LIN {X 0,Y 178.864,Z 372.474,A -85,B 0,C 180,E1 -23549.283,E2 -23549.283} C_VEL
LIN {X 0,Y 171.89,Z 372.083,A -85,B 0,C 180,E1 -23553.272,E2 -23553.272} C_VEL
LIN {X 0,Y 166.102,Z 370.53,A -85,B 0,C 180,E1 -23557.617,E2 -23557.617} C_VEL
LIN {X 0,Y 161.684,Z 367.817,A -85,B 0,C 180,E1 -23562.286,E2 -23562.286} C_VEL
LIN {X 0,Y 158.988,Z 364.935,A -85,B 0,C 180,E1 -23565.929,E2 -23565.929} C_VEL
LIN {X 0,Y 156.894,Z 359.998,A -85,B 0,C 180,E1 -23570.999,E2 -23570.999} C_VEL
LIN {X 0,Y 156.126,Z 355.356,A -85,B 0,C 180,E1 -23574.835,E2 -23574.835} C_VEL
LIN {X 0,Y 155.711,Z 348.695,A -85,B 0,C 180,E1 -23579.354,E2 -23579.354} C_VEL
LIN {X 0,Y 155.836,Z 341.725,A -85,B 0,C 180,E1 -23583.232,E2 -23583.232} C_VEL
LIN {X 0,Y 156.247,Z 333.011,A -85,B 0,C 180,E1 -23587.197,E2 -23587.197} C_VEL
LIN {X 0,Y 157.032,Z 322.982,A -85,B 0,C 180,E1 -23590.965,E2 -23590.965} C_VEL
LIN {X 0,Y 158.084,Z 311.456,A -85,B 0,C 180,E1 -23594.482,E2 -23594.482} C_VEL
LIN {X 0,Y 159.277,Z 300.027,A -85,B 0,C 180,E1 -23597.328,E2 -23597.328} C_VEL
LIN {X 0,Y 160.585,Z 287.52,A -85,B 0,C 180,E1 -23599.827,E2 -23599.827} C_VEL
LIN {X 0,Y 159.751,Z 280.238,A -85,B 0,C 180,E1 -23601.02,E2 -23601.02} C_VEL
LIN {X 0,Y 158.066,Z 266.61,A -85,B 0,C 180,E1 -23602.867,E2 -23602.867} C_VEL
LIN {X 0,Y 157.49,Z 258.741,A -85,B 0,C 180,E1 -23603.767,E2 -23603.767} C_VEL
LIN {X 0,Y 158.382,Z 249.573,A -85,B 0,C 180,E1 -23609.948,E2 -23609.948} C_VEL
LIN {X 0,Y 159.359,Z 242.124,A -85,B 0,C 180,E1 -23614.982,E2 -23614.982} C_VEL
LIN {X 0,Y 159.793,Z 237.68,A -85,B 0,C 180,E1 -23618.007,E2 -23618.007} C_VEL
LIN {X 0,Y 159.018,Z 232.396,A -85,B 0,C 180,E1 -23621.843,E2 -23621.843} C_VEL
LIN {X 0,Y 159.402,Z 233.851,A -85,B 0,C 180,E1 -23625.131,E2 -23625.131} C_VEL
LIN {X 0,Y 159.637,Z 235.642,A -85,B 0,C 180,E1 -23628.668,E2 -23628.668} C_VEL
LIN {X 0,Y 160.053,Z 238.877,A -85,B 0,C 180,E1 -23634.376,E2 -23634.376} C_VEL
LIN {X 0,Y 161.694,Z 242.388,A -85,B 0,C 180,E1 -23635.252,E2 -23635.252} C_VEL
LIN {X 0,Y 165.253,Z 249.918,A -85,B 0,C 180,E1 -23637.133,E2 -23637.133} C_VEL
LIN {X 0,Y 167.935,Z 257.855,A -85,B 0,C 180,E1 -23639.086,E2 -23639.086} C_VEL
LIN {X 0,Y 169.717,Z 265.352,A -85,B 0,C 180,E1 -23641.054,E2 -23641.054} C_VEL
LIN {X 0,Y 170.772,Z 272.517,A -85,B 0,C 180,E1 -23643.08,E2 -23643.08} C_VEL
LIN {X 0,Y 171.198,Z 278.169,A -85,B 0,C 180,E1 -23644.84,E2 -23644.84} C_VEL
LIN {X 0,Y 170.665,Z 280.993,A -85,B 0,C 180,E1 -23645.679,E2 -23645.679} C_VEL
LIN {X 0,Y 167.855,Z 289.578,A -85,B 0,C 180,E1 -23648.506,E2 -23648.506} C_VEL
LIN {X 0,Y 165.094,Z 296.179,A -85,B 0,C 180,E1 -23651.378,E2 -23651.378} C_VEL
LIN {X 0,Y 163.429,Z 300.329,A -85,B 0,C 180,E1 -23653.765,E2 -23653.765} C_VEL
LIN {X 0,Y 161.928,Z 303.706,A -85,B 0,C 180,E1 -23656.186,E2 -23656.186} C_VEL
LIN {X 0,Y 160.418,Z 307.486,A -85,B 0,C 180,E1 -23659.904,E2 -23659.904} C_VEL
LIN {X 0,Y 159.37,Z 309.319,A -85,B 0,C 180,E1 -23662.394,E2 -23662.394} C_VEL
LIN {X 0,Y 158.847,Z 310.546,A -85,B 0,C 180,E1 -23664.92,E2 -23664.92} C_VEL
LIN {X 0,Y 158.433,Z 311.303,A -85,B 0,C 180,E1 -23667.454,E2 -23667.454} C_VEL
LIN {X 0,Y 158.279,Z 311.577,A -85,B 0,C 180,E1 -23669.997,E2 -23669.997} C_VEL
LIN {X 0,Y 158.432,Z 311.335,A -85,B 0,C 180,E1 -23672.539,E2 -23672.539} C_VEL
LIN {X 0,Y 158.845,Z 310.622,A -85,B 0,C 180,E1 -23675.073,E2 -23675.073} C_VEL
LIN {X 0,Y 159.367,Z 309.426,A -85,B 0,C 180,E1 -23677.599,E2 -23677.599} C_VEL
LIN {X 0,Y 160.955,Z 306.53,A -85,B 0,C 180,E1 -23681.328,E2 -23681.328} C_VEL
LIN {X 0,Y 162.457,Z 302.377,A -85,B 0,C 180,E1 -23685.041,E2 -23685.041} C_VEL
LIN {X 0,Y 163.482,Z 300.591,A -85,B 0,C 180,E1 -23686.223,E2 -23686.223} C_VEL
LIN {X 0,Y 165.079,Z 296.507,A -85,B 0,C 180,E1 -23688.617,E2 -23688.617} C_VEL
LIN {X 0,Y 167.817,Z 289.962,A -85,B 0,C 180,E1 -23691.493,E2 -23691.493} C_VEL
LIN {X 0,Y 170.602,Z 281.568,A -85,B 0,C 180,E1 -23694.324,E2 -23694.324} C_VEL
LIN {X 0,Y 171.271,Z 277.73,A -85,B 0,C 180,E1 -23695.476,E2 -23695.476} C_VEL
LIN {X 0,Y 170.427,Z 269.133,A -85,B 0,C 180,E1 -23698.096,E2 -23698.096} C_VEL
LIN {X 0,Y 168.581,Z 260.042,A -85,B 0,C 180,E1 -23700.542,E2 -23700.542} C_VEL
LIN {X 0,Y 165.775,Z 251.147,A -85,B 0,C 180,E1 -23702.753,E2 -23702.753} C_VEL
LIN {X 0,Y 161.837,Z 242.466,A -85,B 0,C 180,E1 -23704.901,E2 -23704.901} C_VEL
LIN {X 0,Y 160.31,Z 239.516,A -85,B 0,C 180,E1 -23705.627,E2 -23705.627} C_VEL
LIN {X 0,Y 160.14,Z 238.936,A -85,B 0,C 180,E1 -23705.743,E2 -23705.743} C_VEL
LIN {X 0,Y 159.65,Z 235.706,A -85,B 0,C 180,E1 -23711.551,E2 -23711.551} C_VEL
LIN {X 0,Y 159.33,Z 233.908,A -85,B 0,C 180,E1 -23715.109,E2 -23715.109} C_VEL
LIN {X 0,Y 159.092,Z 232.317,A -85,B 0,C 180,E1 -23718.67,E2 -23718.67} C_VEL
LIN {X 0,Y 158.736,Z 230.624,A -85,B 0,C 180,E1 -23722.833,E2 -23722.833} C_VEL
LIN {X 0,Y 158.461,Z 228.914,A -85,B 0,C 180,E1 -23727.844,E2 -23727.844} C_VEL
LIN {X 0,Y 158.156,Z 227.327,A -85,B 0,C 180,E1 -23733.617,E2 -23733.617} C_VEL
LIN {X 0,Y 157.925,Z 226.263,A -85,B 0,C 180,E1 -23739.144,E2 -23739.144} C_VEL
LIN {X 0,Y 157.872,Z 225.638,A -85,B 0,C 180,E1 -23744.508,E2 -23744.508} C_VEL
LIN {X 0,Y 158.084,Z 225.448,A -85,B 0,C 180,E1 -23749.756,E2 -23749.756} C_VEL
LIN {X 0,Y 158.195,Z 225.509,A -85,B 0,C 180,E1 -23752.341,E2 -23752.341} C_VEL
LIN {X 0,Y 158.794,Z 226.144,A -85,B 0,C 180,E1 -23760,E2 -23760} C_VEL
LIN {X 0,Y 158.687,Z 227.58,A -85,B 0,C 180,E1 -23765.082,E2 -23765.082} C_VEL
LIN {X 0,Y 159.105,Z 229.328,A -85,B 0,C 180,E1 -23770.177,E2 -23770.177} C_VEL
LIN {X 0,Y 159.387,Z 231.672,A -85,B 0,C 180,E1 -23775.341,E2 -23775.341} C_VEL
LIN {X 0,Y 159.941,Z 234.494,A -85,B 0,C 180,E1 -23780.581,E2 -23780.581} C_VEL
LIN {X 0,Y 160.713,Z 237.968,A -85,B 0,C 180,E1 -23785.932,E2 -23785.932} C_VEL
LIN {X 0,Y 161.422,Z 240.536,A -85,B 0,C 180,E1 -23789.46,E2 -23789.46} C_VEL
LIN {X 0,Y 162.358,Z 244.484,A -85,B 0,C 180,E1 -23794.245,E2 -23794.245} C_VEL
LIN {X 0,Y 163.242,Z 249.108,A -85,B 0,C 180,E1 -23799.206,E2 -23799.206} C_VEL
LIN {X 0,Y 164.036,Z 253.296,A -85,B 0,C 180,E1 -23803.276,E2 -23803.276} C_VEL
LIN {X 0,Y 165.228,Z 258.701,A -85,B 0,C 180,E1 -23808.211,E2 -23808.211} C_VEL
LIN {X 0,Y 165.717,Z 261.5,A -85,B 0,C 180,E1 -23810.491,E2 -23810.491} C_VEL
LIN {X 0,Y 167.275,Z 265.557,A -85,B 0,C 180,E1 -23811.212,E2 -23811.212} C_VEL
LIN {X 0,Y 167.835,Z 268.967,A -85,B 0,C 180,E1 -23811.673,E2 -23811.673} C_VEL
LIN {X 0,Y 168.302,Z 280.321,A -85,B 0,C 180,E1 -23813.191,E2 -23813.191} C_VEL
LIN {X 0,Y 167.94,Z 290.791,A -85,B 0,C 180,E1 -23814.876,E2 -23814.876} C_VEL
LIN {X 0,Y 166.952,Z 302.091,A -85,B 0,C 180,E1 -23817.146,E2 -23817.146} C_VEL
LIN {X 0,Y 165.032,Z 313.463,A -85,B 0,C 180,E1 -23819.979,E2 -23819.979} C_VEL
LIN {X 0,Y 163.62,Z 321.527,A -85,B 0,C 180,E1 -23822.504,E2 -23822.504} C_VEL
LIN {X 0,Y 162.576,Z 326.775,A -85,B 0,C 180,E1 -23824.391,E2 -23824.391} C_VEL
LIN {X 0,Y 159.816,Z 335.261,A -85,B 0,C 180,E1 -23828.075,E2 -23828.075} C_VEL
LIN {X 0,Y 157.929,Z 341.848,A -85,B 0,C 180,E1 -23831.854,E2 -23831.854} C_VEL
LIN {X 0,Y 156.88,Z 347.042,A -85,B 0,C 180,E1 -23835.739,E2 -23835.739} C_VEL
LIN {X 0,Y 156.611,Z 350.924,A -85,B 0,C 180,E1 -23839.663,E2 -23839.663} C_VEL
LIN {X 0,Y 156.875,Z 352.842,A -85,B 0,C 180,E1 -23842.28,E2 -23842.28} C_VEL
LIN {X 0,Y 157.572,Z 354.473,A -85,B 0,C 180,E1 -23845.046,E2 -23845.046} C_VEL
LIN {X 0,Y 157.668,Z 360.13,A -85,B 0,C 180,E1 -23848.088,E2 -23848.088} C_VEL
LIN {X 0,Y 157.721,Z 364.985,A -85,B 0,C 180,E1 -23851.28,E2 -23851.28} C_VEL
LIN {X 0,Y 157.19,Z 368.04,A -85,B 0,C 180,E1 -23853.849,E2 -23853.849} C_VEL
LIN {X 0,Y 156.604,Z 372.902,A -85,B 0,C 180,E1 -23859.139,E2 -23859.139} C_VEL
LIN {X 0,Y 157.016,Z 375.5,A -85,B 0,C 180,E1 -23862.936,E2 -23862.936} C_VEL
LIN {X 0,Y 158.818,Z 378.029,A -85,B 0,C 180,E1 -23868.048,E2 -23868.048} C_VEL
LIN {X 0,Y 162.378,Z 379.502,A -85,B 0,C 180,E1 -23872.929,E2 -23872.929} C_VEL
LIN {X 0,Y 167.343,Z 379.897,A -85,B 0,C 180,E1 -23877.518,E2 -23877.518} C_VEL
LIN {X 0,Y 173.897,Z 379.136,A -85,B 0,C 180,E1 -23882.062,E2 -23882.062} C_VEL
LIN {X 0,Y 176.385,Z 378.542,A -85,B 0,C 180,E1 -23883.806,E2 -23883.806} C_VEL
LIN {X 0,Y 182.265,Z 376.171,A -85,B 0,C 180,E1 -23889.128,E2 -23889.128} C_VEL
LIN {X 0,Y 185.289,Z 375.099,A -85,B 0,C 180,E1 -23890.661,E2 -23890.661} C_VEL
LIN {X 0,Y 186.544,Z 374.692,A -85,B 0,C 180,E1 -23891.107,E2 -23891.107} C_VEL
LIN {X 0,Y 196.969,Z 371.002,A -85,B 0,C 180,E1 -23894.092,E2 -23894.092} C_VEL
LIN {X 0,Y 206.383,Z 366.992,A -85,B 0,C 180,E1 -23896.276,E2 -23896.276} C_VEL
LIN {X 0,Y 206.868,Z 366.673,A -85,B 0,C 180,E1 -23896.802,E2 -23896.802} C_VEL
LIN {X 0,Y 195.531,Z 370.197,A -85,B 0,C 180,E1 -23899.686,E2 -23899.686} C_VEL
LIN {X 0,Y 185.739,Z 372.251,A -85,B 0,C 180,E1 -23902.742,E2 -23902.742} C_VEL
LIN {X 0,Y 176.867,Z 373.129,A -85,B 0,C 180,E1 -23906.199,E2 -23906.199} C_VEL
LIN {X 0,Y 169.061,Z 372.868,A -85,B 0,C 180,E1 -23910.076,E2 -23910.076} C_VEL
LIN {X 0,Y 162.472,Z 371.472,A -85,B 0,C 180,E1 -23914.369,E2 -23914.369} C_VEL
LIN {X 0,Y 157.09,Z 368.939,A -85,B 0,C 180,E1 -23919.028,E2 -23919.028} C_VEL
LIN {X 0,Y 153.921,Z 366.285,A -85,B 0,C 180,E1 -23922.735,E2 -23922.735} C_VEL
LIN {X 0,Y 150.781,Z 361.312,A -85,B 0,C 180,E1 -23928.201,E2 -23928.201} C_VEL
LIN {X 0,Y 149.417,Z 355.617,A -85,B 0,C 180,E1 -23933.247,E2 -23933.247} C_VEL
LIN {X 0,Y 148.823,Z 349.002,A -85,B 0,C 180,E1 -23937.97,E2 -23937.97} C_VEL
LIN {X 0,Y 148.897,Z 342.118,A -85,B 0,C 180,E1 -23942.029,E2 -23942.029} C_VEL
LIN {X 0,Y 149.262,Z 332.846,A -85,B 0,C 180,E1 -23946.469,E2 -23946.469} C_VEL
LIN {X 0,Y 149.939,Z 323.553,A -85,B 0,C 180,E1 -23950.143,E2 -23950.143} C_VEL
LIN {X 0,Y 150.875,Z 312.241,A -85,B 0,C 180,E1 -23953.812,E2 -23953.812} C_VEL
LIN {X 0,Y 152.079,Z 301.001,A -85,B 0,C 180,E1 -23956.788,E2 -23956.788} C_VEL
LIN {X 0,Y 153.295,Z 288.755,A -85,B 0,C 180,E1 -23959.414,E2 -23959.414} C_VEL
LIN {X 0,Y 153.455,Z 286.043,A -85,B 0,C 180,E1 -23959.915,E2 -23959.915} C_VEL
LIN {X 0,Y 151.644,Z 272.518,A -85,B 0,C 180,E1 -23962.035,E2 -23962.035} C_VEL
LIN {X 0,Y 150.41,Z 259.023,A -85,B 0,C 180,E1 -23963.766,E2 -23963.766} C_VEL
LIN {X 0,Y 151.428,Z 249.075,A -85,B 0,C 180,E1 -23970.699,E2 -23970.699} C_VEL
LIN {X 0,Y 152.459,Z 241.499,A -85,B 0,C 180,E1 -23975.997,E2 -23975.997} C_VEL
LIN {X 0,Y 152.707,Z 237.915,A -85,B 0,C 180,E1 -23978.516,E2 -23978.516} C_VEL
LIN {X 0,Y 152.184,Z 234.339,A -85,B 0,C 180,E1 -23981.251,E2 -23981.251} C_VEL
LIN {X 0,Y 152.521,Z 235.356,A -85,B 0,C 180,E1 -23983.724,E2 -23983.724} C_VEL
LIN {X 0,Y 152.726,Z 237.106,A -85,B 0,C 180,E1 -23987.415,E2 -23987.415} C_VEL
LIN {X 0,Y 153.074,Z 239.709,A -85,B 0,C 180,E1 -23992.366,E2 -23992.366} C_VEL
LIN {X 0,Y 154.668,Z 242.942,A -85,B 0,C 180,E1 -23993.207,E2 -23993.207} C_VEL
LIN {X 0,Y 155.811,Z 245.048,A -85,B 0,C 180,E1 -23993.797,E2 -23993.797} C_VEL
LIN {X 0,Y 159.269,Z 252.262,A -85,B 0,C 180,E1 -23995.829,E2 -23995.829} C_VEL
LIN {X 0,Y 161.81,Z 259.863,A -85,B 0,C 180,E1 -23997.885,E2 -23997.885} C_VEL
LIN {X 0,Y 163.406,Z 266.927,A -85,B 0,C 180,E1 -23999.893,E2 -23999.893} C_VEL
LIN {X 0,Y 164.382,Z 273.706,A -85,B 0,C 180,E1 -24001.943,E2 -24001.943} C_VEL
LIN {X 0,Y 164.742,Z 279.468,A -85,B 0,C 180,E1 -24003.845,E2 -24003.845} C_VEL
LIN {X 0,Y 164.297,Z 282.089,A -85,B 0,C 180,E1 -24004.671,E2 -24004.671} C_VEL
LIN {X 0,Y 161.344,Z 290.607,A -85,B 0,C 180,E1 -24007.592,E2 -24007.592} C_VEL
LIN {X 0,Y 158.451,Z 297.187,A -85,B 0,C 180,E1 -24010.567,E2 -24010.567} C_VEL
LIN {X 0,Y 156.69,Z 301.324,A -85,B 0,C 180,E1 -24013.046,E2 -24013.046} C_VEL
LIN {X 0,Y 155.112,Z 304.69,A -85,B 0,C 180,E1 -24015.566,E2 -24015.566} C_VEL
LIN {X 0,Y 153.503,Z 308.463,A -85,B 0,C 180,E1 -24019.444,E2 -24019.444} C_VEL
LIN {X 0,Y 152.407,Z 310.294,A -85,B 0,C 180,E1 -24022.045,E2 -24022.045} C_VEL
LIN {X 0,Y 151.848,Z 311.521,A -85,B 0,C 180,E1 -24024.685,E2 -24024.685} C_VEL
LIN {X 0,Y 151.412,Z 312.277,A -85,B 0,C 180,E1 -24027.336,E2 -24027.336} C_VEL
LIN {X 0,Y 151.252,Z 312.551,A -85,B 0,C 180,E1 -24029.997,E2 -24029.997} C_VEL
LIN {X 0,Y 151.411,Z 312.308,A -85,B 0,C 180,E1 -24032.657,E2 -24032.657} C_VEL
LIN {X 0,Y 151.846,Z 311.595,A -85,B 0,C 180,E1 -24035.308,E2 -24035.308} C_VEL
LIN {X 0,Y 152.404,Z 310.399,A -85,B 0,C 180,E1 -24037.948,E2 -24037.948} C_VEL
LIN {X 0,Y 154.069,Z 307.506,A -85,B 0,C 180,E1 -24041.842,E2 -24041.842} C_VEL
LIN {X 0,Y 155.678,Z 303.363,A -85,B 0,C 180,E1 -24045.712,E2 -24045.712} C_VEL
LIN {X 0,Y 156.745,Z 301.581,A -85,B 0,C 180,E1 -24046.941,E2 -24046.941} C_VEL
LIN {X 0,Y 158.436,Z 297.507,A -85,B 0,C 180,E1 -24049.428,E2 -24049.428} C_VEL
LIN {X 0,Y 161.306,Z 290.98,A -85,B 0,C 180,E1 -24052.406,E2 -24052.406} C_VEL
LIN {X 0,Y 164.238,Z 282.656,A -85,B 0,C 180,E1 -24055.332,E2 -24055.332} C_VEL
LIN {X 0,Y 164.832,Z 279.138,A -85,B 0,C 180,E1 -24056.442,E2 -24056.442} C_VEL
LIN {X 0,Y 164.087,Z 270.378,A -85,B 0,C 180,E1 -24059.284,E2 -24059.284} C_VEL
LIN {X 0,Y 162.45,Z 262.158,A -85,B 0,C 180,E1 -24061.663,E2 -24061.663} C_VEL
LIN {X 0,Y 159.924,Z 253.695,A -85,B 0,C 180,E1 -24063.955,E2 -24063.955} C_VEL
LIN {X 0,Y 156.36,Z 245.98,A -85,B 0,C 180,E1 -24066.127,E2 -24066.127} C_VEL
LIN {X 0,Y 154.786,Z 243.034,A -85,B 0,C 180,E1 -24066.961,E2 -24066.961} C_VEL
LIN {X 0,Y 153.226,Z 240.057,A -85,B 0,C 180,E1 -24067.771,E2 -24067.771} C_VEL
LIN {X 0,Y 153.127,Z 239.728,A -85,B 0,C 180,E1 -24067.834,E2 -24067.834} C_VEL
LIN {X 0,Y 152.637,Z 236.782,A -85,B 0,C 180,E1 -24073.677,E2 -24073.677} C_VEL
LIN {X 0,Y 152.362,Z 234.975,A -85,B 0,C 180,E1 -24077.558,E2 -24077.558} C_VEL
LIN {X 0,Y 152.003,Z 232.845,A -85,B 0,C 180,E1 -24083.053,E2 -24083.053} C_VEL
LIN {X 0,Y 151.779,Z 231.712,A -85,B 0,C 180,E1 -24086.45,E2 -24086.45} C_VEL
LIN {X 0,Y 151.526,Z 230.067,A -85,B 0,C 180,E1 -24092.366,E2 -24092.366} C_VEL
LIN {X 0,Y 151.309,Z 228.984,A -85,B 0,C 180,E1 -24098.263,E2 -24098.263} C_VEL
LIN {X 0,Y 151.254,Z 228.312,A -85,B 0,C 180,E1 -24103.812,E2 -24103.812} C_VEL
LIN {X 0,Y 151.448,Z 228.042,A -85,B 0,C 180,E1 -24109.302,E2 -24109.302} C_VEL
LIN {X 0,Y 151.56,Z 228.118,A -85,B 0,C 180,E1 -24112.003,E2 -24112.003} C_VEL
LIN {X 0,Y 152.238,Z 228.866,A -85,B 0,C 180,E1 -24120,E2 -24120} C_VEL
LIN {X 0,Y 152.318,Z 231.152,A -85,B 0,C 180,E1 -24127.956,E2 -24127.956} C_VEL
LIN {X 0,Y 152.516,Z 232.117,A -85,B 0,C 180,E1 -24130.622,E2 -24130.622} C_VEL
LIN {X 0,Y 152.791,Z 234.571,A -85,B 0,C 180,E1 -24136.021,E2 -24136.021} C_VEL
LIN {X 0,Y 153.395,Z 237.585,A -85,B 0,C 180,E1 -24141.502,E2 -24141.502} C_VEL
LIN {X 0,Y 154.228,Z 241.192,A -85,B 0,C 180,E1 -24147.109,E2 -24147.109} C_VEL
LIN {X 0,Y 154.88,Z 243.62,A -85,B 0,C 180,E1 -24150.447,E2 -24150.447} C_VEL
LIN {X 0,Y 155.641,Z 246.736,A -85,B 0,C 180,E1 -24154.313,E2 -24154.313} C_VEL
LIN {X 0,Y 156.394,Z 250.891,A -85,B 0,C 180,E1 -24158.986,E2 -24158.986} C_VEL
LIN {X 0,Y 157.405,Z 256.254,A -85,B 0,C 180,E1 -24164.412,E2 -24164.412} C_VEL
LIN {X 0,Y 158.394,Z 260.751,A -85,B 0,C 180,E1 -24168.481,E2 -24168.481} C_VEL
LIN {X 0,Y 159.977,Z 264.664,A -85,B 0,C 180,E1 -24169.272,E2 -24169.272} C_VEL
LIN {X 0,Y 161.904,Z 269.992,A -85,B 0,C 180,E1 -24170.338,E2 -24170.338} C_VEL
LIN {X 0,Y 162.183,Z 281.863,A -85,B 0,C 180,E1 -24172.067,E2 -24172.067} C_VEL
LIN {X 0,Y 161.538,Z 293.013,A -85,B 0,C 180,E1 -24174.036,E2 -24174.036} C_VEL
LIN {X 0,Y 160.337,Z 303.73,A -85,B 0,C 180,E1 -24176.39,E2 -24176.39} C_VEL
LIN {X 0,Y 158.499,Z 313.385,A -85,B 0,C 180,E1 -24178.976,E2 -24178.976} C_VEL
LIN {X 0,Y 157.083,Z 320.419,A -85,B 0,C 180,E1 -24181.256,E2 -24181.256} C_VEL
LIN {X 0,Y 156.074,Z 325.715,A -85,B 0,C 180,E1 -24183.241,E2 -24183.241} C_VEL
LIN {X 0,Y 153.58,Z 332.999,A -85,B 0,C 180,E1 -24186.456,E2 -24186.456} C_VEL
LIN {X 0,Y 151.418,Z 339.86,A -85,B 0,C 180,E1 -24190.34,E2 -24190.34} C_VEL
LIN {X 0,Y 150.203,Z 344.463,A -85,B 0,C 180,E1 -24193.699,E2 -24193.699} C_VEL
LIN {X 0,Y 149.568,Z 348.753,A -85,B 0,C 180,E1 -24197.796,E2 -24197.796} C_VEL
LIN {X 0,Y 149.749,Z 351.845,A -85,B 0,C 180,E1 -24201.91,E2 -24201.91} C_VEL
LIN {X 0,Y 150.845,Z 354.08,A -85,B 0,C 180,E1 -24206.163,E2 -24206.163} C_VEL
LIN {X 0,Y 151.002,Z 360.641,A -85,B 0,C 180,E1 -24210.003,E2 -24210.003} C_VEL
LIN {X 0,Y 150.832,Z 364.278,A -85,B 0,C 180,E1 -24212.674,E2 -24212.674} C_VEL
LIN {X 0,Y 149.863,Z 369.751,A -85,B 0,C 180,E1 -24218.091,E2 -24218.091} C_VEL
LIN {X 0,Y 150.284,Z 373.803,A -85,B 0,C 180,E1 -24223.526,E2 -24223.526} C_VEL
LIN {X 0,Y 152.208,Z 376.635,A -85,B 0,C 180,E1 -24228.861,E2 -24228.861} C_VEL
LIN {X 0,Y 155.915,Z 378.43,A -85,B 0,C 180,E1 -24233.937,E2 -24233.937} C_VEL
LIN {X 0,Y 161.093,Z 379.187,A -85,B 0,C 180,E1 -24238.682,E2 -24238.682} C_VEL
LIN {X 0,Y 167.79,Z 378.872,A -85,B 0,C 180,E1 -24243.266,E2 -24243.266} C_VEL
LIN {X 0,Y 175.313,Z 377.662,A -85,B 0,C 180,E1 -24246.968,E2 -24246.968} C_VEL
LIN {X 0,Y 184.37,Z 375.373,A -85,B 0,C 180,E1 -24250.396,E2 -24250.396} C_VEL
LIN {X 0,Y 186.544,Z 374.692,A -85,B 0,C 180,E1 -24251.107,E2 -24251.107} C_VEL
LIN {X 0,Y 189.607,Z 373.61,A -85,B 0,C 180,E1 -24252.382,E2 -24252.382} C_VEL
LIN {X 0,Y 191.844,Z 372.609,A -85,B 0,C 180,E1 -24253.805,E2 -24253.805} C_VEL
LIN {X 0,Y 195.424,Z 370.753,A -85,B 0,C 180,E1 -24256.797,E2 -24256.797} C_VEL
LIN {X 0,Y 195.624,Z 370.657,A -85,B 0,C 180,E1 -24256.953,E2 -24256.953} C_VEL
LIN {X 0,Y 185.126,Z 372.791,A -85,B 0,C 180,E1 -24259.806,E2 -24259.806} C_VEL
LIN {X 0,Y 175.508,Z 373.778,A -85,B 0,C 180,E1 -24263.083,E2 -24263.083} C_VEL
LIN {X 0,Y 166.879,Z 373.642,A -85,B 0,C 180,E1 -24266.805,E2 -24266.805} C_VEL
LIN {X 0,Y 159.371,Z 372.382,A -85,B 0,C 180,E1 -24270.982,E2 -24270.982} C_VEL
LIN {X 0,Y 153.106,Z 370.012,A -85,B 0,C 180,E1 -24275.599,E2 -24275.599} C_VEL
LIN {X 0,Y 148.317,Z 366.524,A -85,B 0,C 180,E1 -24280.628,E2 -24280.628} C_VEL
LIN {X 0,Y 145.4,Z 363.116,A -85,B 0,C 180,E1 -24284.583,E2 -24284.583} C_VEL
LIN {X 0,Y 143.037,Z 356.88,A -85,B 0,C 180,E1 -24290.575,E2 -24290.575} C_VEL
LIN {X 0,Y 142.135,Z 350.231,A -85,B 0,C 180,E1 -24295.747,E2 -24295.747} C_VEL
LIN {X 0,Y 141.995,Z 342.388,A -85,B 0,C 180,E1 -24300.709,E2 -24300.709} C_VEL
LIN {X 0,Y 142.184,Z 334.091,A -85,B 0,C 180,E1 -24304.962,E2 -24304.962} C_VEL
LIN {X 0,Y 142.843,Z 324.084,A -85,B 0,C 180,E1 -24309.202,E2 -24309.202} C_VEL
LIN {X 0,Y 143.643,Z 314.039,A -85,B 0,C 180,E1 -24312.719,E2 -24312.719} C_VEL
LIN {X 0,Y 144.864,Z 301.779,A -85,B 0,C 180,E1 -24316.198,E2 -24316.198} C_VEL
LIN {X 0,Y 146.088,Z 289.833,A -85,B 0,C 180,E1 -24318.949,E2 -24318.949} C_VEL
LIN {X 0,Y 146.267,Z 285.301,A -85,B 0,C 180,E1 -24319.835,E2 -24319.835} C_VEL
LIN {X 0,Y 144.263,Z 270.23,A -85,B 0,C 180,E1 -24322.231,E2 -24322.231} C_VEL
LIN {X 0,Y 143.341,Z 259.378,A -85,B 0,C 180,E1 -24323.668,E2 -24323.668} C_VEL
LIN {X 0,Y 144.49,Z 248.507,A -85,B 0,C 180,E1 -24331.526,E2 -24331.526} C_VEL
LIN {X 0,Y 145.54,Z 240.76,A -85,B 0,C 180,E1 -24337.129,E2 -24337.129} C_VEL
LIN {X 0,Y 145.427,Z 236.854,A -85,B 0,C 180,E1 -24340.027,E2 -24340.027} C_VEL
LIN {X 0,Y 145.35,Z 236.313,A -85,B 0,C 180,E1 -24340.471,E2 -24340.471} C_VEL
LIN {X 0,Y 145.773,Z 237.522,A -85,B 0,C 180,E1 -24343.678,E2 -24343.678} C_VEL
LIN {X 0,Y 146.052,Z 240.273,A -85,B 0,C 180,E1 -24349.531,E2 -24349.531} C_VEL
LIN {X 0,Y 146.106,Z 240.609,A -85,B 0,C 180,E1 -24350.014,E2 -24350.014} C_VEL
LIN {X 0,Y 147.613,Z 243.668,A -85,B 0,C 180,E1 -24350.9,E2 -24350.9} C_VEL
LIN {X 0,Y 148.999,Z 245.812,A -85,B 0,C 180,E1 -24351.649,E2 -24351.649} C_VEL
LIN {X 0,Y 152.407,Z 252.608,A -85,B 0,C 180,E1 -24353.8,E2 -24353.8} C_VEL
LIN {X 0,Y 155.214,Z 260.043,A -85,B 0,C 180,E1 -24356.06,E2 -24356.06} C_VEL
LIN {X 0,Y 156.963,Z 267.387,A -85,B 0,C 180,E1 -24358.291,E2 -24358.291} C_VEL
LIN {X 0,Y 157.869,Z 273.196,A -85,B 0,C 180,E1 -24360.129,E2 -24360.129} C_VEL
LIN {X 0,Y 158.361,Z 280.231,A -85,B 0,C 180,E1 -24362.573,E2 -24362.573} C_VEL
LIN {X 0,Y 157.999,Z 283.18,A -85,B 0,C 180,E1 -24363.585,E2 -24363.585} C_VEL
LIN {X 0,Y 154.879,Z 291.636,A -85,B 0,C 180,E1 -24366.603,E2 -24366.603} C_VEL
LIN {X 0,Y 151.843,Z 298.194,A -85,B 0,C 180,E1 -24369.684,E2 -24369.684} C_VEL
LIN {X 0,Y 149.978,Z 302.319,A -85,B 0,C 180,E1 -24372.263,E2 -24372.263} C_VEL
LIN {X 0,Y 148.314,Z 305.674,A -85,B 0,C 180,E1 -24374.89,E2 -24374.89} C_VEL
LIN {X 0,Y 146.6,Z 309.438,A -85,B 0,C 180,E1 -24378.941,E2 -24378.941} C_VEL
LIN {X 0,Y 145.45,Z 311.27,A -85,B 0,C 180,E1 -24381.662,E2 -24381.662} C_VEL
LIN {X 0,Y 144.852,Z 312.494,A -85,B 0,C 180,E1 -24384.428,E2 -24384.428} C_VEL
LIN {X 0,Y 144.392,Z 313.25,A -85,B 0,C 180,E1 -24387.207,E2 -24387.207} C_VEL
LIN {X 0,Y 144.224,Z 313.525,A -85,B 0,C 180,E1 -24389.996,E2 -24389.996} C_VEL
LIN {X 0,Y 144.391,Z 313.282,A -85,B 0,C 180,E1 -24392.786,E2 -24392.786} C_VEL
LIN {X 0,Y 144.85,Z 312.569,A -85,B 0,C 180,E1 -24395.565,E2 -24395.565} C_VEL
LIN {X 0,Y 145.447,Z 311.372,A -85,B 0,C 180,E1 -24398.331,E2 -24398.331} C_VEL
LIN {X 0,Y 147.197,Z 308.483,A -85,B 0,C 180,E1 -24402.403,E2 -24402.403} C_VEL
LIN {X 0,Y 148.923,Z 304.349,A -85,B 0,C 180,E1 -24406.445,E2 -24406.445} C_VEL
LIN {X 0,Y 150.035,Z 302.569,A -85,B 0,C 180,E1 -24407.723,E2 -24407.723} C_VEL
LIN {X 0,Y 151.829,Z 298.504,A -85,B 0,C 180,E1 -24410.31,E2 -24410.31} C_VEL
LIN {X 0,Y 154.84,Z 291.997,A -85,B 0,C 180,E1 -24413.396,E2 -24413.396} C_VEL
LIN {X 0,Y 157.926,Z 283.744,A -85,B 0,C 180,E1 -24416.421,E2 -24416.421} C_VEL
LIN {X 0,Y 158.346,Z 282.149,A -85,B 0,C 180,E1 -24416.91,E2 -24416.91} C_VEL
LIN {X 0,Y 158.141,Z 275.539,A -85,B 0,C 180,E1 -24419.261,E2 -24419.261} C_VEL
LIN {X 0,Y 157.141,Z 267.705,A -85,B 0,C 180,E1 -24421.814,E2 -24421.814} C_VEL
LIN {X 0,Y 155.235,Z 259.921,A -85,B 0,C 180,E1 -24424.169,E2 -24424.169} C_VEL
LIN {X 0,Y 152.025,Z 251.531,A -85,B 0,C 180,E1 -24426.714,E2 -24426.714} C_VEL
LIN {X 0,Y 148.335,Z 244.538,A -85,B 0,C 180,E1 -24428.964,E2 -24428.964} C_VEL
LIN {X 0,Y 146.503,Z 241.661,A -85,B 0,C 180,E1 -24429.968,E2 -24429.968} C_VEL
LIN {X 0,Y 146.11,Z 240.498,A -85,B 0,C 180,E1 -24430.298,E2 -24430.298} C_VEL
LIN {X 0,Y 145.889,Z 238.898,A -85,B 0,C 180,E1 -24433.73,E2 -24433.73} C_VEL
LIN {X 0,Y 145.64,Z 237.221,A -85,B 0,C 180,E1 -24437.5,E2 -24437.5} C_VEL
LIN {X 0,Y 145.385,Z 235.838,A -85,B 0,C 180,E1 -24441.065,E2 -24441.065} C_VEL
LIN {X 0,Y 145.1,Z 234.424,A -85,B 0,C 180,E1 -24445.42,E2 -24445.42} C_VEL
LIN {X 0,Y 144.864,Z 232.845,A -85,B 0,C 180,E1 -24450.978,E2 -24450.978} C_VEL
LIN {X 0,Y 144.74,Z 232.177,A -85,B 0,C 180,E1 -24454.087,E2 -24454.087} C_VEL
LIN {X 0,Y 144.605,Z 231.271,A -85,B 0,C 180,E1 -24460.11,E2 -24460.11} C_VEL
LIN {X 0,Y 144.719,Z 230.808,A -85,B 0,C 180,E1 -24466.213,E2 -24466.213} C_VEL
LIN {X 0,Y 144.939,Z 230.753,A -85,B 0,C 180,E1 -24471.635,E2 -24471.635} C_VEL
LIN {X 0,Y 145.287,Z 231.236,A -85,B 0,C 180,E1 -24477.227,E2 -24477.227} C_VEL
LIN {X 0,Y 145.696,Z 231.631,A -85,B 0,C 180,E1 -24480,E2 -24480} C_VEL
LIN {X 0,Y 145.58,Z 233.124,A -85,B 0,C 180,E1 -24485.541,E2 -24485.541} C_VEL
LIN {X 0,Y 145.928,Z 235.003,A -85,B 0,C 180,E1 -24491.107,E2 -24491.107} C_VEL
LIN {X 0,Y 146.209,Z 237.525,A -85,B 0,C 180,E1 -24496.763,E2 -24496.763} C_VEL
LIN {X 0,Y 146.829,Z 240.634,A -85,B 0,C 180,E1 -24502.515,E2 -24502.515} C_VEL
LIN {X 0,Y 147.796,Z 244.397,A -85,B 0,C 180,E1 -24508.393,E2 -24508.393} C_VEL
LIN {X 0,Y 148.64,Z 247.741,A -85,B 0,C 180,E1 -24512.937,E2 -24512.937} C_VEL
LIN {X 0,Y 149.376,Z 251.731,A -85,B 0,C 180,E1 -24517.708,E2 -24517.708} C_VEL
LIN {X 0,Y 150.208,Z 256.333,A -85,B 0,C 180,E1 -24522.731,E2 -24522.731} C_VEL
LIN {X 0,Y 150.873,Z 259.711,A -85,B 0,C 180,E1 -24526.125,E2 -24526.125} C_VEL
LIN {X 0,Y 152.421,Z 263.519,A -85,B 0,C 180,E1 -24526.982,E2 -24526.982} C_VEL
LIN {X 0,Y 153.694,Z 266.125,A -85,B 0,C 180,E1 -24527.641,E2 -24527.641} C_VEL
LIN {X 0,Y 156.096,Z 272.227,A -85,B 0,C 180,E1 -24529.088,E2 -24529.088} C_VEL
LIN {X 0,Y 156.111,Z 283.75,A -85,B 0,C 180,E1 -24530.935,E2 -24530.935} C_VEL
LIN {X 0,Y 155.157,Z 295.149,A -85,B 0,C 180,E1 -24533.147,E2 -24533.147} C_VEL
LIN {X 0,Y 153.912,Z 304.089,A -85,B 0,C 180,E1 -24535.278,E2 -24535.278} C_VEL
LIN {X 0,Y 152.252,Z 312.247,A -85,B 0,C 180,E1 -24537.551,E2 -24537.551} C_VEL
LIN {X 0,Y 150.65,Z 319.314,A -85,B 0,C 180,E1 -24539.905,E2 -24539.905} C_VEL
LIN {X 0,Y 149.149,Z 326.156,A -85,B 0,C 180,E1 -24542.654,E2 -24542.654} C_VEL
LIN {X 0,Y 146.771,Z 332.665,A -85,B 0,C 180,E1 -24545.7,E2 -24545.7} C_VEL
LIN {X 0,Y 144.652,Z 338.843,A -85,B 0,C 180,E1 -24549.379,E2 -24549.379} C_VEL
LIN {X 0,Y 143.298,Z 343.456,A -85,B 0,C 180,E1 -24552.89,E2 -24552.89} C_VEL
LIN {X 0,Y 142.536,Z 347.753,A -85,B 0,C 180,E1 -24557.184,E2 -24557.184} C_VEL
LIN {X 0,Y 142.631,Z 350.847,A -85,B 0,C 180,E1 -24561.503,E2 -24561.503} C_VEL
LIN {X 0,Y 143.886,Z 353.035,A -85,B 0,C 180,E1 -24566.503,E2 -24566.503} C_VEL
LIN {X 0,Y 144.145,Z 353.27,A -85,B 0,C 180,E1 -24567.209,E2 -24567.209} C_VEL
LIN {X 0,Y 144.303,Z 359.984,A -85,B 0,C 180,E1 -24571.399,E2 -24571.399} C_VEL
LIN {X 0,Y 143.825,Z 363.4,A -85,B 0,C 180,E1 -24574.207,E2 -24574.207} C_VEL
LIN {X 0,Y 143.151,Z 368.436,A -85,B 0,C 180,E1 -24579.482,E2 -24579.482} C_VEL
LIN {X 0,Y 143.614,Z 371.919,A -85,B 0,C 180,E1 -24584.167,E2 -24584.167} C_VEL
LIN {X 0,Y 145.65,Z 375.059,A -85,B 0,C 180,E1 -24589.745,E2 -24589.745} C_VEL
LIN {X 0,Y 149.533,Z 377.184,A -85,B 0,C 180,E1 -24595.028,E2 -24595.028} C_VEL
LIN {X 0,Y 154.929,Z 378.298,A -85,B 0,C 180,E1 -24599.937,E2 -24599.937} C_VEL
LIN {X 0,Y 161.564,Z 378.42,A -85,B 0,C 180,E1 -24604.44,E2 -24604.44} C_VEL
LIN {X 0,Y 169.707,Z 377.595,A -85,B 0,C 180,E1 -24608.406,E2 -24608.406} C_VEL
LIN {X 0,Y 179.037,Z 375.768,A -85,B 0,C 180,E1 -24611.865,E2 -24611.865} C_VEL
LIN {X 0,Y 189.273,Z 372.928,A -85,B 0,C 180,E1 -24614.873,E2 -24614.873} C_VEL
LIN {X 0,Y 194.698,Z 371.11,A -85,B 0,C 180,E1 -24616.218,E2 -24616.218} C_VEL
LIN {X 0,Y 195.424,Z 370.753,A -85,B 0,C 180,E1 -24616.797,E2 -24616.797} C_VEL
LIN {X 0,Y 195.424,Z 370.637,A -85,B 0,C 180,E1 -24617.344,E2 -24617.344} C_VEL
LIN {X 0,Y 193.79,Z 370.967,A -85,B 0,C 180,E1 -24618.147,E2 -24618.147} C_VEL
LIN {X 0,Y 189.729,Z 371.895,A -85,B 0,C 180,E1 -24619.004,E2 -24619.004} C_VEL
LIN {X 0,Y 186.249,Z 372.606,A -85,B 0,C 180,E1 -24619.447,E2 -24619.447} C_VEL
LIN {X 0,Y 174.759,Z 374.286,A -85,B 0,C 180,E1 -24620.648,E2 -24620.648} C_VEL
LIN {X 0,Y 170.688,Z 374.508,A -85,B 0,C 180,E1 -24621.465,E2 -24621.465} C_VEL
LIN {X 0,Y 168.967,Z 374.5,A -85,B 0,C 180,E1 -24622.017,E2 -24622.017} C_VEL
LIN {X 0,Y 160.988,Z 373.942,A -85,B 0,C 180,E1 -24625.423,E2 -24625.423} C_VEL
LIN {X 0,Y 153.205,Z 372.267,A -85,B 0,C 180,E1 -24629.695,E2 -24629.695} C_VEL
LIN {X 0,Y 146.701,Z 369.507,A -85,B 0,C 180,E1 -24634.459,E2 -24634.459} C_VEL
LIN {X 0,Y 141.694,Z 365.631,A -85,B 0,C 180,E1 -24639.684,E2 -24639.684} C_VEL
LIN {X 0,Y 138.68,Z 361.908,A -85,B 0,C 180,E1 -24643.816,E2 -24643.816} C_VEL
LIN {X 0,Y 136.352,Z 355.871,A -85,B 0,C 180,E1 -24649.607,E2 -24649.607} C_VEL
LIN {X 0,Y 135.378,Z 349.311,A -85,B 0,C 180,E1 -24654.788,E2 -24654.788} C_VEL
LIN {X 0,Y 135.152,Z 341.261,A -85,B 0,C 180,E1 -24660,E2 -24660} C_VEL
LIN {X 0,Y 135.306,Z 332.826,A -85,B 0,C 180,E1 -24664.469,E2 -24664.469} C_VEL
LIN {X 0,Y 135.945,Z 322.602,A -85,B 0,C 180,E1 -24668.922,E2 -24668.922} C_VEL
LIN {X 0,Y 136.783,Z 311.906,A -85,B 0,C 180,E1 -24672.725,E2 -24672.725} C_VEL
LIN {X 0,Y 137.987,Z 299.702,A -85,B 0,C 180,E1 -24676.268,E2 -24676.268} C_VEL
LIN {X 0,Y 139.221,Z 287.239,A -85,B 0,C 180,E1 -24679.155,E2 -24679.155} C_VEL
LIN {X 0,Y 138.632,Z 281.653,A -85,B 0,C 180,E1 -24680.204,E2 -24680.204} C_VEL
LIN {X 0,Y 136.846,Z 267.587,A -85,B 0,C 180,E1 -24682.409,E2 -24682.409} C_VEL
LIN {X 0,Y 136.251,Z 259.856,A -85,B 0,C 180,E1 -24683.424,E2 -24683.424} C_VEL
LIN {X 0,Y 137.384,Z 248.925,A -85,B 0,C 180,E1 -24691.625,E2 -24691.625} C_VEL
LIN {X 0,Y 138.346,Z 242.611,A -85,B 0,C 180,E1 -24696.373,E2 -24696.373} C_VEL
LIN {X 0,Y 138.464,Z 238.315,A -85,B 0,C 180,E1 -24699.659,E2 -24699.659} C_VEL
LIN {X 0,Y 139.062,Z 240.32,A -85,B 0,C 180,E1 -24705.036,E2 -24705.036} C_VEL
LIN {X 0,Y 139.2,Z 241.424,A -85,B 0,C 180,E1 -24707.333,E2 -24707.333} C_VEL
LIN {X 0,Y 140.638,Z 244.433,A -85,B 0,C 180,E1 -24708.296,E2 -24708.296} C_VEL
LIN {X 0,Y 141.999,Z 246.369,A -85,B 0,C 180,E1 -24709.106,E2 -24709.106} C_VEL
LIN {X 0,Y 145.481,Z 252.701,A -85,B 0,C 180,E1 -24711.438,E2 -24711.438} C_VEL
LIN {X 0,Y 148.65,Z 260.386,A -85,B 0,C 180,E1 -24714.063,E2 -24714.063} C_VEL
LIN {X 0,Y 150.493,Z 267.501,A -85,B 0,C 180,E1 -24716.408,E2 -24716.408} C_VEL
LIN {X 0,Y 151.633,Z 274.932,A -85,B 0,C 180,E1 -24718.948,E2 -24718.948} C_VEL
LIN {X 0,Y 151.969,Z 281.786,A -85,B 0,C 180,E1 -24721.484,E2 -24721.484} C_VEL
LIN {X 0,Y 151.751,Z 284.274,A -85,B 0,C 180,E1 -24722.407,E2 -24722.407} C_VEL
LIN {X 0,Y 148.463,Z 292.666,A -85,B 0,C 180,E1 -24725.527,E2 -24725.527} C_VEL
LIN {X 0,Y 145.274,Z 299.199,A -85,B 0,C 180,E1 -24728.722,E2 -24728.722} C_VEL
LIN {X 0,Y 143.298,Z 303.313,A -85,B 0,C 180,E1 -24731.407,E2 -24731.407} C_VEL
LIN {X 0,Y 141.54,Z 306.659,A -85,B 0,C 180,E1 -24734.148,E2 -24734.148} C_VEL
LIN {X 0,Y 139.709,Z 310.413,A -85,B 0,C 180,E1 -24738.388,E2 -24738.388} C_VEL
LIN {X 0,Y 138.5,Z 312.245,A -85,B 0,C 180,E1 -24741.24,E2 -24741.24} C_VEL
LIN {X 0,Y 137.859,Z 313.469,A -85,B 0,C 180,E1 -24744.144,E2 -24744.144} C_VEL
LIN {X 0,Y 137.373,Z 314.224,A -85,B 0,C 180,E1 -24747.064,E2 -24747.064} C_VEL
LIN {X 0,Y 137.196,Z 314.5,A -85,B 0,C 180,E1 -24749.996,E2 -24749.996} C_VEL
LIN {X 0,Y 137.372,Z 314.256,A -85,B 0,C 180,E1 -24752.929,E2 -24752.929} C_VEL
LIN {X 0,Y 137.857,Z 313.543,A -85,B 0,C 180,E1 -24755.848,E2 -24755.848} C_VEL
LIN {X 0,Y 138.497,Z 312.345,A -85,B 0,C 180,E1 -24758.753,E2 -24758.753} C_VEL
LIN {X 0,Y 140.34,Z 309.46,A -85,B 0,C 180,E1 -24763.02,E2 -24763.02} C_VEL
LIN {X 0,Y 142.194,Z 305.335,A -85,B 0,C 180,E1 -24767.247,E2 -24767.247} C_VEL
LIN {X 0,Y 143.356,Z 303.557,A -85,B 0,C 180,E1 -24768.578,E2 -24768.578} C_VEL
LIN {X 0,Y 145.26,Z 299.501,A -85,B 0,C 180,E1 -24771.272,E2 -24771.272} C_VEL
LIN {X 0,Y 148.424,Z 293.015,A -85,B 0,C 180,E1 -24774.472,E2 -24774.472} C_VEL
LIN {X 0,Y 151.676,Z 284.83,A -85,B 0,C 180,E1 -24777.6,E2 -24777.6} C_VEL
LIN {X 0,Y 152.045,Z 282.122,A -85,B 0,C 180,E1 -24778.569,E2 -24778.569} C_VEL
LIN {X 0,Y 151.703,Z 275.182,A -85,B 0,C 180,E1 -24781.158,E2 -24781.158} C_VEL
LIN {X 0,Y 150.697,Z 268.132,A -85,B 0,C 180,E1 -24783.597,E2 -24783.597} C_VEL
LIN {X 0,Y 149.003,Z 261.178,A -85,B 0,C 180,E1 -24785.869,E2 -24785.869} C_VEL
LIN {X 0,Y 145.845,Z 253.208,A -85,B 0,C 180,E1 -24788.57,E2 -24788.57} C_VEL
LIN {X 0,Y 141.299,Z 245.258,A -85,B 0,C 180,E1 -24791.566,E2 -24791.566} C_VEL
LIN {X 0,Y 139.486,Z 242.34,A -85,B 0,C 180,E1 -24792.696,E2 -24792.696} C_VEL
LIN {X 0,Y 139.131,Z 241.334,A -85,B 0,C 180,E1 -24793.04,E2 -24793.04} C_VEL
LIN {X 0,Y 138.728,Z 238.764,A -85,B 0,C 180,E1 -24799.449,E2 -24799.449} C_VEL
LIN {X 0,Y 138.461,Z 237.096,A -85,B 0,C 180,E1 -24804.297,E2 -24804.297} C_VEL
LIN {X 0,Y 138.192,Z 235.586,A -85,B 0,C 180,E1 -24809.824,E2 -24809.824} C_VEL
LIN {X 0,Y 138.04,Z 234.405,A -85,B 0,C 180,E1 -24815.964,E2 -24815.964} C_VEL
LIN {X 0,Y 137.951,Z 233.596,A -85,B 0,C 180,E1 -24822.201,E2 -24822.201} C_VEL
LIN {X 0,Y 138.205,Z 233.375,A -85,B 0,C 180,E1 -24828.263,E2 -24828.263} C_VEL
LIN {X 0,Y 138.324,Z 233.421,A -85,B 0,C 180,E1 -24831.232,E2 -24831.232} C_VEL
LIN {X 0,Y 138.686,Z 233.871,A -85,B 0,C 180,E1 -24837.095,E2 -24837.095} C_VEL
LIN {X 0,Y 139.082,Z 234.269,A -85,B 0,C 180,E1 -24840,E2 -24840} C_VEL
LIN {X 0,Y 139.004,Z 235.837,A -85,B 0,C 180,E1 -24845.804,E2 -24845.804} C_VEL
LIN {X 0,Y 139.326,Z 237.82,A -85,B 0,C 180,E1 -24851.64,E2 -24851.64} C_VEL
LIN {X 0,Y 139.583,Z 240.142,A -85,B 0,C 180,E1 -24856.947,E2 -24856.947} C_VEL
LIN {X 0,Y 139.923,Z 242.02,A -85,B 0,C 180,E1 -24860.585,E2 -24860.585} C_VEL
LIN {X 0,Y 140.745,Z 245.653,A -85,B 0,C 180,E1 -24866.706,E2 -24866.706} C_VEL
LIN {X 0,Y 141.323,Z 247.681,A -85,B 0,C 180,E1 -24869.822,E2 -24869.822} C_VEL
LIN {X 0,Y 142.121,Z 251.255,A -85,B 0,C 180,E1 -24874.659,E2 -24874.659} C_VEL
LIN {X 0,Y 142.85,Z 255.489,A -85,B 0,C 180,E1 -24879.761,E2 -24879.761} C_VEL
LIN {X 0,Y 143.529,Z 259.017,A -85,B 0,C 180,E1 -24883.518,E2 -24883.518} C_VEL
LIN {X 0,Y 145.1,Z 262.797,A -85,B 0,C 180,E1 -24884.491,E2 -24884.491} C_VEL
LIN {X 0,Y 146.333,Z 265.119,A -85,B 0,C 180,E1 -24885.186,E2 -24885.186} C_VEL
LIN {X 0,Y 148.861,Z 271.003,A -85,B 0,C 180,E1 -24886.8,E2 -24886.8} C_VEL
LIN {X 0,Y 150.271,Z 274.684,A -85,B 0,C 180,E1 -24887.778,E2 -24887.778} C_VEL
LIN {X 0,Y 150.016,Z 286.053,A -85,B 0,C 180,E1 -24889.823,E2 -24889.823} C_VEL
LIN {X 0,Y 148.813,Z 296.954,A -85,B 0,C 180,E1 -24892.129,E2 -24892.129} C_VEL
LIN {X 0,Y 147.257,Z 305.944,A -85,B 0,C 180,E1 -24894.483,E2 -24894.483} C_VEL
LIN {X 0,Y 145.045,Z 315.34,A -85,B 0,C 180,E1 -24897.386,E2 -24897.386} C_VEL
LIN {X 0,Y 142.709,Z 325.094,A -85,B 0,C 180,E1 -24901.309,E2 -24901.309} C_VEL
LIN {X 0,Y 140.632,Z 330.887,A -85,B 0,C 180,E1 -24904.098,E2 -24904.098} C_VEL
LIN {X 0,Y 137.942,Z 337.828,A -85,B 0,C 180,E1 -24908.327,E2 -24908.327} C_VEL
LIN {X 0,Y 136.428,Z 342.448,A -85,B 0,C 180,E1 -24912,E2 -24912} C_VEL
LIN {X 0,Y 135.517,Z 346.751,A -85,B 0,C 180,E1 -24916.508,E2 -24916.508} C_VEL
LIN {X 0,Y 135.52,Z 349.849,A -85,B 0,C 180,E1 -24921.054,E2 -24921.054} C_VEL
LIN {X 0,Y 136.034,Z 351.295,A -85,B 0,C 180,E1 -24924.073,E2 -24924.073} C_VEL
LIN {X 0,Y 137.497,Z 352.659,A -85,B 0,C 180,E1 -24928.539,E2 -24928.539} C_VEL
LIN {X 0,Y 137.643,Z 357.204,A -85,B 0,C 180,E1 -24931.467,E2 -24931.467} C_VEL
LIN {X 0,Y 137.56,Z 359.177,A -85,B 0,C 180,E1 -24932.932,E2 -24932.932} C_VEL
LIN {X 0,Y 136.557,Z 365.245,A -85,B 0,C 180,E1 -24938.886,E2 -24938.886} C_VEL
LIN {X 0,Y 137.026,Z 369.886,A -85,B 0,C 180,E1 -24944.863,E2 -24944.863} C_VEL
LIN {X 0,Y 139.17,Z 373.341,A -85,B 0,C 180,E1 -24950.705,E2 -24950.705} C_VEL
LIN {X 0,Y 143.261,Z 375.797,A -85,B 0,C 180,E1 -24956.204,E2 -24956.204} C_VEL
LIN {X 0,Y 148.885,Z 377.255,A -85,B 0,C 180,E1 -24961.285,E2 -24961.285} C_VEL
LIN {X 0,Y 155.782,Z 377.751,A -85,B 0,C 180,E1 -24965.912,E2 -24965.912} C_VEL
LIN {X 0,Y 164.227,Z 377.349,A -85,B 0,C 180,E1 -24969.938,E2 -24969.938} C_VEL
LIN {X 0,Y 173.828,Z 375.983,A -85,B 0,C 180,E1 -24973.422,E2 -24973.422} C_VEL
LIN {X 0,Y 184.332,Z 373.633,A -85,B 0,C 180,E1 -24976.423,E2 -24976.423} C_VEL
LIN {X 0,Y 185.104,Z 373.363,A -85,B 0,C 180,E1 -24976.888,E2 -24976.888} C_VEL
LIN {X 0,Y 174.774,Z 374.415,A -85,B 0,C 180,E1 -24979.955,E2 -24979.955} C_VEL
LIN {X 0,Y 168.967,Z 374.5,A -85,B 0,C 180,E1 -24982.017,E2 -24982.017} C_VEL
LIN {X 0,Y 164.656,Z 374.412,A -85,B 0,C 180,E1 -24983.406,E2 -24983.406} C_VEL
LIN {X 0,Y 156.559,Z 373.747,A -85,B 0,C 180,E1 -24985.439,E2 -24985.439} C_VEL
LIN {X 0,Y 148.892,Z 372.386,A -85,B 0,C 180,E1 -24987.717,E2 -24987.717} C_VEL
LIN {X 0,Y 145.352,Z 371.223,A -85,B 0,C 180,E1 -24989.493,E2 -24989.493} C_VEL
LIN {X 0,Y 140.365,Z 368.786,A -85,B 0,C 180,E1 -24993.216,E2 -24993.216} C_VEL
LIN {X 0,Y 135.153,Z 364.55,A -85,B 0,C 180,E1 -24998.654,E2 -24998.654} C_VEL
LIN {X 0,Y 132.023,Z 360.517,A -85,B 0,C 180,E1 -25002.976,E2 -25002.976} C_VEL
LIN {X 0,Y 129.589,Z 354.109,A -85,B 0,C 180,E1 -25009.058,E2 -25009.058} C_VEL
LIN {X 0,Y 128.577,Z 347.204,A -85,B 0,C 180,E1 -25014.511,E2 -25014.511} C_VEL
LIN {X 0,Y 128.377,Z 338.717,A -85,B 0,C 180,E1 -25020,E2 -25020} C_VEL
LIN {X 0,Y 128.552,Z 329.793,A -85,B 0,C 180,E1 -25024.704,E2 -25024.704} C_VEL
LIN {X 0,Y 129.218,Z 318.993,A -85,B 0,C 180,E1 -25029.391,E2 -25029.391} C_VEL
LIN {X 0,Y 130.244,Z 306.43,A -85,B 0,C 180,E1 -25033.749,E2 -25033.749} C_VEL
LIN {X 0,Y 131.465,Z 294.403,A -85,B 0,C 180,E1 -25037.099,E2 -25037.099} C_VEL
LIN {X 0,Y 132.112,Z 285.07,A -85,B 0,C 180,E1 -25039.218,E2 -25039.218} C_VEL
LIN {X 0,Y 130.227,Z 271.638,A -85,B 0,C 180,E1 -25041.571,E2 -25041.571} C_VEL
LIN {X 0,Y 129.175,Z 260.17,A -85,B 0,C 180,E1 -25043.239,E2 -25043.239} C_VEL
LIN {X 0,Y 130.171,Z 249.997,A -85,B 0,C 180,E1 -25051.204,E2 -25051.204} C_VEL
LIN {X 0,Y 131.282,Z 243.108,A -85,B 0,C 180,E1 -25056.576,E2 -25056.576} C_VEL
LIN {X 0,Y 131.515,Z 240.404,A -85,B 0,C 180,E1 -25058.726,E2 -25058.726} C_VEL
LIN {X 0,Y 132.013,Z 241.344,A -85,B 0,C 180,E1 -25061.808,E2 -25061.808} C_VEL
LIN {X 0,Y 132.279,Z 242.406,A -85,B 0,C 180,E1 -25064.222,E2 -25064.222} C_VEL
LIN {X 0,Y 134.251,Z 245.878,A -85,B 0,C 180,E1 -25065.657,E2 -25065.657} C_VEL
LIN {X 0,Y 135.432,Z 247.61,A -85,B 0,C 180,E1 -25066.462,E2 -25066.462} C_VEL
LIN {X 0,Y 139.691,Z 255.37,A -85,B 0,C 180,E1 -25069.694,E2 -25069.694} C_VEL
LIN {X 0,Y 142.826,Z 263.031,A -85,B 0,C 180,E1 -25072.633,E2 -25072.633} C_VEL
LIN {X 0,Y 144.521,Z 269.878,A -85,B 0,C 180,E1 -25075.148,E2 -25075.148} C_VEL
LIN {X 0,Y 145.318,Z 275.46,A -85,B 0,C 180,E1 -25077.188,E2 -25077.188} C_VEL
LIN {X 0,Y 145.666,Z 281.57,A -85,B 0,C 180,E1 -25079.56,E2 -25079.56} C_VEL
LIN {X 0,Y 145.549,Z 285.372,A -85,B 0,C 180,E1 -25081.124,E2 -25081.124} C_VEL
LIN {X 0,Y 142.104,Z 293.696,A -85,B 0,C 180,E1 -25084.354,E2 -25084.354} C_VEL
LIN {X 0,Y 138.75,Z 300.203,A -85,B 0,C 180,E1 -25087.669,E2 -25087.669} C_VEL
LIN {X 0,Y 136.653,Z 304.307,A -85,B 0,C 180,E1 -25090.467,E2 -25090.467} C_VEL
LIN {X 0,Y 134.792,Z 307.644,A -85,B 0,C 180,E1 -25093.332,E2 -25093.332} C_VEL
LIN {X 0,Y 132.832,Z 311.389,A -85,B 0,C 180,E1 -25097.778,E2 -25097.778} C_VEL
LIN {X 0,Y 131.559,Z 313.219,A -85,B 0,C 180,E1 -25100.774,E2 -25100.774} C_VEL
LIN {X 0,Y 130.87,Z 314.444,A -85,B 0,C 180,E1 -25103.83,E2 -25103.83} C_VEL
LIN {X 0,Y 130.355,Z 315.198,A -85,B 0,C 180,E1 -25106.905,E2 -25106.905} C_VEL
LIN {X 0,Y 130.168,Z 315.474,A -85,B 0,C 180,E1 -25109.996,E2 -25109.996} C_VEL
LIN {X 0,Y 130.354,Z 315.229,A -85,B 0,C 180,E1 -25113.087,E2 -25113.087} C_VEL
LIN {X 0,Y 130.868,Z 314.517,A -85,B 0,C 180,E1 -25116.162,E2 -25116.162} C_VEL
LIN {X 0,Y 131.555,Z 313.318,A -85,B 0,C 180,E1 -25119.218,E2 -25119.218} C_VEL
LIN {X 0,Y 133.502,Z 310.435,A -85,B 0,C 180,E1 -25123.699,E2 -25123.699} C_VEL
LIN {X 0,Y 135.495,Z 306.319,A -85,B 0,C 180,E1 -25128.128,E2 -25128.128} C_VEL
LIN {X 0,Y 136.712,Z 304.544,A -85,B 0,C 180,E1 -25129.517,E2 -25129.517} C_VEL
LIN {X 0,Y 138.736,Z 300.496,A -85,B 0,C 180,E1 -25132.325,E2 -25132.325} C_VEL
LIN {X 0,Y 142.065,Z 294.032,A -85,B 0,C 180,E1 -25135.645,E2 -25135.645} C_VEL
LIN {X 0,Y 145.491,Z 285.911,A -85,B 0,C 180,E1 -25138.881,E2 -25138.881} C_VEL
LIN {X 0,Y 145.76,Z 282.07,A -85,B 0,C 180,E1 -25140.417,E2 -25140.417} C_VEL
LIN {X 0,Y 145.224,Z 273.446,A -85,B 0,C 180,E1 -25143.774,E2 -25143.774} C_VEL
LIN {X 0,Y 143.908,Z 266.478,A -85,B 0,C 180,E1 -25146.309,E2 -25146.309} C_VEL
LIN {X 0,Y 141.453,Z 259.102,A -85,B 0,C 180,E1 -25149.053,E2 -25149.053} C_VEL
LIN {X 0,Y 137.373,Z 250.833,A -85,B 0,C 180,E1 -25152.383,E2 -25152.383} C_VEL
LIN {X 0,Y 135.324,Z 247.389,A -85,B 0,C 180,E1 -25153.883,E2 -25153.883} C_VEL
LIN {X 0,Y 132.479,Z 243.194,A -85,B 0,C 180,E1 -25155.857,E2 -25155.857} C_VEL
LIN {X 0,Y 132.133,Z 242.236,A -85,B 0,C 180,E1 -25156.254,E2 -25156.254} C_VEL
LIN {X 0,Y 131.93,Z 240.79,A -85,B 0,C 180,E1 -25160.264,E2 -25160.264} C_VEL
LIN {X 0,Y 131.796,Z 239.556,A -85,B 0,C 180,E1 -25164.085,E2 -25164.085} C_VEL
LIN {X 0,Y 131.52,Z 238.308,A -85,B 0,C 180,E1 -25168.75,E2 -25168.75} C_VEL
LIN {X 0,Y 131.377,Z 237.121,A -85,B 0,C 180,E1 -25174.662,E2 -25174.662} C_VEL
LIN {X 0,Y 131.347,Z 236.367,A -85,B 0,C 180,E1 -25181.274,E2 -25181.274} C_VEL
LIN {X 0,Y 131.541,Z 235.981,A -85,B 0,C 180,E1 -25187.66,E2 -25187.66} C_VEL
LIN {X 0,Y 131.687,Z 236.016,A -85,B 0,C 180,E1 -25190.787,E2 -25190.787} C_VEL
LIN {X 0,Y 132.097,Z 236.533,A -85,B 0,C 180,E1 -25196.95,E2 -25196.95} C_VEL
LIN {X 0,Y 132.476,Z 236.924,A -85,B 0,C 180,E1 -25200,E2 -25200} C_VEL
LIN {X 0,Y 132.397,Z 238.545,A -85,B 0,C 180,E1 -25206.094,E2 -25206.094} C_VEL
LIN {X 0,Y 132.562,Z 239.51,A -85,B 0,C 180,E1 -25209.152,E2 -25209.152} C_VEL
LIN {X 0,Y 132.708,Z 240.648,A -85,B 0,C 180,E1 -25212.23,E2 -25212.23} C_VEL
LIN {X 0,Y 133.021,Z 243.429,A -85,B 0,C 180,E1 -25218.482,E2 -25218.482} C_VEL
LIN {X 0,Y 133.741,Z 246.84,A -85,B 0,C 180,E1 -25224.859,E2 -25224.859} C_VEL
LIN {X 0,Y 134.58,Z 249.842,A -85,B 0,C 180,E1 -25229.743,E2 -25229.743} C_VEL
LIN {X 0,Y 135.336,Z 253.44,A -85,B 0,C 180,E1 -25234.836,E2 -25234.836} C_VEL
LIN {X 0,Y 136.161,Z 258.052,A -85,B 0,C 180,E1 -25240.456,E2 -25240.456} C_VEL
LIN {X 0,Y 137.913,Z 262.143,A -85,B 0,C 180,E1 -25241.681,E2 -25241.681} C_VEL
LIN {X 0,Y 139.07,Z 264.151,A -85,B 0,C 180,E1 -25242.404,E2 -25242.404} C_VEL
LIN {X 0,Y 143.203,Z 273.651,A -85,B 0,C 180,E1 -25245.367,E2 -25245.367} C_VEL
LIN {X 0,Y 144.612,Z 277.639,A -85,B 0,C 180,E1 -25246.548,E2 -25246.548} C_VEL
LIN {X 0,Y 143.891,Z 288.503,A -85,B 0,C 180,E1 -25248.669,E2 -25248.669} C_VEL
LIN {X 0,Y 142.251,Z 299.996,A -85,B 0,C 180,E1 -25251.385,E2 -25251.385} C_VEL
LIN {X 0,Y 140.061,Z 309.968,A -85,B 0,C 180,E1 -25254.32,E2 -25254.32} C_VEL
LIN {X 0,Y 138.099,Z 317.114,A -85,B 0,C 180,E1 -25256.838,E2 -25256.838} C_VEL
LIN {X 0,Y 136.252,Z 324.016,A -85,B 0,C 180,E1 -25259.812,E2 -25259.812} C_VEL
LIN {X 0,Y 134.343,Z 329.533,A -85,B 0,C 180,E1 -25262.577,E2 -25262.577} C_VEL
LIN {X 0,Y 131.297,Z 336.814,A -85,B 0,C 180,E1 -25267.17,E2 -25267.17} C_VEL
LIN {X 0,Y 129.604,Z 341.442,A -85,B 0,C 180,E1 -25271.017,E2 -25271.017} C_VEL
LIN {X 0,Y 128.541,Z 345.753,A -85,B 0,C 180,E1 -25275.761,E2 -25275.761} C_VEL
LIN {X 0,Y 128.403,Z 348.849,A -85,B 0,C 180,E1 -25280.553,E2 -25280.553} C_VEL
LIN {X 0,Y 128.882,Z 350.298,A -85,B 0,C 180,E1 -25283.743,E2 -25283.743} C_VEL
LIN {X 0,Y 130.656,Z 351.593,A -85,B 0,C 180,E1 -25289.233,E2 -25289.233} C_VEL
LIN {X 0,Y 130.93,Z 351.937,A -85,B 0,C 180,E1 -25290.004,E2 -25290.004} C_VEL
LIN {X 0,Y 130.988,Z 356.325,A -85,B 0,C 180,E1 -25293.08,E2 -25293.08} C_VEL
LIN {X 0,Y 130.132,Z 361.333,A -85,B 0,C 180,E1 -25297.764,E2 -25297.764} C_VEL
LIN {X 0,Y 130.144,Z 366.253,A -85,B 0,C 180,E1 -25303.583,E2 -25303.583} C_VEL
LIN {X 0,Y 131.392,Z 369.72,A -85,B 0,C 180,E1 -25308.723,E2 -25308.723} C_VEL
LIN {X 0,Y 134.677,Z 372.969,A -85,B 0,C 180,E1 -25314.679,E2 -25314.679} C_VEL
LIN {X 0,Y 139.789,Z 375.255,A -85,B 0,C 180,E1 -25320.187,E2 -25320.187} C_VEL
LIN {X 0,Y 147.165,Z 376.681,A -85,B 0,C 180,E1 -25325.723,E2 -25325.723} C_VEL
LIN {X 0,Y 154.308,Z 377.018,A -85,B 0,C 180,E1 -25329.62,E2 -25329.62} C_VEL
LIN {X 0,Y 163.662,Z 376.578,A -85,B 0,C 180,E1 -25333.403,E2 -25333.403} C_VEL
LIN {X 0,Y 174.622,Z 375.077,A -85,B 0,C 180,E1 -25336.827,E2 -25336.827} C_VEL
LIN {X 0,Y 163.699,Z 375.039,A -85,B 0,C 180,E1 -25340.391,E2 -25340.391} C_VEL
LIN {X 0,Y 155.199,Z 374.048,A -85,B 0,C 180,E1 -25343.936,E2 -25343.936} C_VEL
LIN {X 0,Y 147.131,Z 371.944,A -85,B 0,C 180,E1 -25348.302,E2 -25348.302} C_VEL
LIN {X 0,Y 145.352,Z 371.223,A -85,B 0,C 180,E1 -25349.493,E2 -25349.493} C_VEL
LIN {X 0,Y 142.056,Z 369.942,A -85,B 0,C 180,E1 -25351.368,E2 -25351.368} C_VEL
LIN {X 0,Y 135.602,Z 367.145,A -85,B 0,C 180,E1 -25354.237,E2 -25354.237} C_VEL
LIN {X 0,Y 130.653,Z 364.408,A -85,B 0,C 180,E1 -25356.653,E2 -25356.653} C_VEL
LIN {X 0,Y 127.768,Z 362.173,A -85,B 0,C 180,E1 -25358.729,E2 -25358.729} C_VEL
LIN {X 0,Y 127.068,Z 361.405,A -85,B 0,C 180,E1 -25359.49,E2 -25359.49} C_VEL
LIN {X 0,Y 123.636,Z 354.867,A -85,B 0,C 180,E1 -25366.005,E2 -25366.005} C_VEL
LIN {X 0,Y 122.067,Z 347.088,A -85,B 0,C 180,E1 -25372.557,E2 -25372.557} C_VEL
LIN {X 0,Y 121.624,Z 338.663,A -85,B 0,C 180,E1 -25378.345,E2 -25378.345} C_VEL
LIN {X 0,Y 121.705,Z 329.838,A -85,B 0,C 180,E1 -25383.311,E2 -25383.311} C_VEL
LIN {X 0,Y 122.236,Z 319.1,A -85,B 0,C 180,E1 -25388.264,E2 -25388.264} C_VEL
LIN {X 0,Y 123.124,Z 307.294,A -85,B 0,C 180,E1 -25392.666,E2 -25392.666} C_VEL
LIN {X 0,Y 124.149,Z 296.404,A -85,B 0,C 180,E1 -25395.977,E2 -25395.977} C_VEL
LIN {X 0,Y 125.117,Z 285.706,A -85,B 0,C 180,E1 -25398.631,E2 -25398.631} C_VEL
LIN {X 0,Y 123.064,Z 270.92,A -85,B 0,C 180,E1 -25401.35,E2 -25401.35} C_VEL
LIN {X 0,Y 122.129,Z 260.506,A -85,B 0,C 180,E1 -25402.957,E2 -25402.957} C_VEL
LIN {X 0,Y 123.168,Z 249.739,A -85,B 0,C 180,E1 -25411.761,E2 -25411.761} C_VEL
LIN {X 0,Y 124.351,Z 242.592,A -85,B 0,C 180,E1 -25417.692,E2 -25417.692} C_VEL
LIN {X 0,Y 125.142,Z 243.222,A -85,B 0,C 180,E1 -25420.361,E2 -25420.361} C_VEL
LIN {X 0,Y 126.863,Z 246.286,A -85,B 0,C 180,E1 -25421.843,E2 -25421.843} C_VEL
LIN {X 0,Y 128.733,Z 248.489,A -85,B 0,C 180,E1 -25423.256,E2 -25423.256} C_VEL
LIN {X 0,Y 131.289,Z 252.883,A -85,B 0,C 180,E1 -25425.408,E2 -25425.408} C_VEL
LIN {X 0,Y 135.527,Z 261.441,A -85,B 0,C 180,E1 -25429.338,E2 -25429.338} C_VEL
LIN {X 0,Y 137.875,Z 268.515,A -85,B 0,C 180,E1 -25432.284,E2 -25432.284} C_VEL
LIN {X 0,Y 139.128,Z 276.192,A -85,B 0,C 180,E1 -25435.34,E2 -25435.34} C_VEL
LIN {X 0,Y 139.467,Z 282.7,A -85,B 0,C 180,E1 -25438.052,E2 -25438.052} C_VEL
LIN {X 0,Y 139.367,Z 286.479,A -85,B 0,C 180,E1 -25439.712,E2 -25439.712} C_VEL
LIN {X 0,Y 135.81,Z 294.725,A -85,B 0,C 180,E1 -25443.072,E2 -25443.072} C_VEL
LIN {X 0,Y 132.277,Z 301.204,A -85,B 0,C 180,E1 -25446.513,E2 -25446.513} C_VEL
LIN {X 0,Y 130.049,Z 305.299,A -85,B 0,C 180,E1 -25449.431,E2 -25449.431} C_VEL
LIN {X 0,Y 128.073,Z 308.628,A -85,B 0,C 180,E1 -25452.43,E2 -25452.43} C_VEL
LIN {X 0,Y 125.972,Z 312.365,A -85,B 0,C 180,E1 -25457.101,E2 -25457.101} C_VEL
LIN {X 0,Y 124.627,Z 314.194,A -85,B 0,C 180,E1 -25460.256,E2 -25460.256} C_VEL
LIN {X 0,Y 123.885,Z 315.419,A -85,B 0,C 180,E1 -25463.481,E2 -25463.481} C_VEL
LIN {X 0,Y 123.338,Z 316.172,A -85,B 0,C 180,E1 -25466.729,E2 -25466.729} C_VEL
LIN {X 0,Y 123.14,Z 316.448,A -85,B 0,C 180,E1 -25469.996,E2 -25469.996} C_VEL
LIN {X 0,Y 123.337,Z 316.203,A -85,B 0,C 180,E1 -25473.262,E2 -25473.262} C_VEL
LIN {X 0,Y 123.883,Z 315.491,A -85,B 0,C 180,E1 -25476.511,E2 -25476.511} C_VEL
LIN {X 0,Y 124.623,Z 314.29,A -85,B 0,C 180,E1 -25479.736,E2 -25479.736} C_VEL
LIN {X 0,Y 126.684,Z 311.412,A -85,B 0,C 180,E1 -25484.452,E2 -25484.452} C_VEL
LIN {X 0,Y 128.832,Z 307.303,A -85,B 0,C 180,E1 -25489.101,E2 -25489.101} C_VEL
LIN {X 0,Y 130.108,Z 305.529,A -85,B 0,C 180,E1 -25490.551,E2 -25490.551} C_VEL
LIN {X 0,Y 132.264,Z 301.492,A -85,B 0,C 180,E1 -25493.481,E2 -25493.481} C_VEL
LIN {X 0,Y 135.77,Z 295.051,A -85,B 0,C 180,E1 -25496.927,E2 -25496.927} C_VEL
LIN {X 0,Y 139.361,Z 286.99,A -85,B 0,C 180,E1 -25500.28,E2 -25500.28} C_VEL
LIN {X 0,Y 139.459,Z 279.116,A -85,B 0,C 180,E1 -25503.661,E2 -25503.661} C_VEL
LIN {X 0,Y 138.754,Z 272.13,A -85,B 0,C 180,E1 -25506.478,E2 -25506.478} C_VEL
LIN {X 0,Y 137.14,Z 265.643,A -85,B 0,C 180,E1 -25509.104,E2 -25509.104} C_VEL
LIN {X 0,Y 134.746,Z 259.549,A -85,B 0,C 180,E1 -25511.737,E2 -25511.737} C_VEL
LIN {X 0,Y 130.577,Z 251.657,A -85,B 0,C 180,E1 -25515.462,E2 -25515.462} C_VEL
LIN {X 0,Y 127.929,Z 247.53,A -85,B 0,C 180,E1 -25517.636,E2 -25517.636} C_VEL
LIN {X 0,Y 125.783,Z 244.613,A -85,B 0,C 180,E1 -25519.361,E2 -25519.361} C_VEL
LIN {X 0,Y 125.218,Z 243.163,A -85,B 0,C 180,E1 -25520.063,E2 -25520.063} C_VEL
LIN {X 0,Y 124.966,Z 241.502,A -85,B 0,C 180,E1 -25525.778,E2 -25525.778} C_VEL
LIN {X 0,Y 124.823,Z 240.622,A -85,B 0,C 180,E1 -25529.553,E2 -25529.553} C_VEL
LIN {X 0,Y 124.755,Z 239.735,A -85,B 0,C 180,E1 -25534.326,E2 -25534.326} C_VEL
LIN {X 0,Y 124.679,Z 238.992,A -85,B 0,C 180,E1 -25540.232,E2 -25540.232} C_VEL
LIN {X 0,Y 124.895,Z 238.698,A -85,B 0,C 180,E1 -25546.992,E2 -25546.992} C_VEL
LIN {X 0,Y 125.061,Z 238.694,A -85,B 0,C 180,E1 -25550.294,E2 -25550.294} C_VEL
LIN {X 0,Y 125.488,Z 239.176,A -85,B 0,C 180,E1 -25556.789,E2 -25556.789} C_VEL
LIN {X 0,Y 125.888,Z 239.621,A -85,B 0,C 180,E1 -25560,E2 -25560} C_VEL
LIN {X 0,Y 125.834,Z 241.321,A -85,B 0,C 180,E1 -25566.413,E2 -25566.413} C_VEL
LIN {X 0,Y 125.984,Z 242.338,A -85,B 0,C 180,E1 -25569.634,E2 -25569.634} C_VEL
LIN {X 0,Y 126.114,Z 243.526,A -85,B 0,C 180,E1 -25572.88,E2 -25572.88} C_VEL
LIN {X 0,Y 126.43,Z 246.387,A -85,B 0,C 180,E1 -25579.483,E2 -25579.483} C_VEL
LIN {X 0,Y 127.257,Z 249.981,A -85,B 0,C 180,E1 -25586.22,E2 -25586.22} C_VEL
LIN {X 0,Y 128.054,Z 253.173,A -85,B 0,C 180,E1 -25591.425,E2 -25591.425} C_VEL
LIN {X 0,Y 128.798,Z 256.929,A -85,B 0,C 180,E1 -25596.803,E2 -25596.803} C_VEL
LIN {X 0,Y 130.431,Z 260.891,A -85,B 0,C 180,E1 -25598.168,E2 -25598.168} C_VEL
LIN {X 0,Y 132.034,Z 263.566,A -85,B 0,C 180,E1 -25599.322,E2 -25599.322} C_VEL
LIN {X 0,Y 134.093,Z 267.934,A -85,B 0,C 180,E1 -25600.93,E2 -25600.93} C_VEL
LIN {X 0,Y 137.91,Z 277.474,A -85,B 0,C 180,E1 -25604.231,E2 -25604.231} C_VEL
LIN {X 0,Y 138.788,Z 280.269,A -85,B 0,C 180,E1 -25605.149,E2 -25605.149} C_VEL
LIN {X 0,Y 137.816,Z 290.697,A -85,B 0,C 180,E1 -25607.398,E2 -25607.398} C_VEL
LIN {X 0,Y 136.059,Z 300.708,A -85,B 0,C 180,E1 -25609.983,E2 -25609.983} C_VEL
LIN {X 0,Y 133.836,Z 309.888,A -85,B 0,C 180,E1 -25612.856,E2 -25612.856} C_VEL
LIN {X 0,Y 131.427,Z 317.799,A -85,B 0,C 180,E1 -25615.847,E2 -25615.847} C_VEL
LIN {X 0,Y 129.46,Z 324.452,A -85,B 0,C 180,E1 -25618.959,E2 -25618.959} C_VEL
LIN {X 0,Y 127.857,Z 328.877,A -85,B 0,C 180,E1 -25621.316,E2 -25621.316} C_VEL
LIN {X 0,Y 124.717,Z 335.799,A -85,B 0,C 180,E1 -25625.891,E2 -25625.891} C_VEL
LIN {X 0,Y 122.833,Z 340.437,A -85,B 0,C 180,E1 -25629.927,E2 -25629.927} C_VEL
LIN {X 0,Y 121.57,Z 344.753,A -85,B 0,C 180,E1 -25634.926,E2 -25634.926} C_VEL
LIN {X 0,Y 121.29,Z 347.892,A -85,B 0,C 180,E1 -25640.079,E2 -25640.079} C_VEL
LIN {X 0,Y 121.74,Z 349.303,A -85,B 0,C 180,E1 -25643.374,E2 -25643.374} C_VEL
LIN {X 0,Y 122.585,Z 350.22,A -85,B 0,C 180,E1 -25646.718,E2 -25646.718} C_VEL
LIN {X 0,Y 124.43,Z 350.784,A -85,B 0,C 180,E1 -25651.42,E2 -25651.42} C_VEL
LIN {X 0,Y 124.497,Z 353.307,A -85,B 0,C 180,E1 -25653.24,E2 -25653.24} C_VEL
LIN {X 0,Y 123.892,Z 356.973,A -85,B 0,C 180,E1 -25656.519,E2 -25656.519} C_VEL
LIN {X 0,Y 123.589,Z 362.914,A -85,B 0,C 180,E1 -25663.152,E2 -25663.152} C_VEL
LIN {X 0,Y 125.004,Z 367.514,A -85,B 0,C 180,E1 -25669.719,E2 -25669.719} C_VEL
LIN {X 0,Y 128.493,Z 371.095,A -85,B 0,C 180,E1 -25675.953,E2 -25675.953} C_VEL
LIN {X 0,Y 133.849,Z 373.699,A -85,B 0,C 180,E1 -25681.677,E2 -25681.677} C_VEL
LIN {X 0,Y 141.662,Z 375.536,A -85,B 0,C 180,E1 -25687.46,E2 -25687.46} C_VEL
LIN {X 0,Y 148.948,Z 376.18,A -85,B 0,C 180,E1 -25691.348,E2 -25691.348} C_VEL
LIN {X 0,Y 158.607,Z 376.165,A -85,B 0,C 180,E1 -25695.156,E2 -25695.156} C_VEL
LIN {X 0,Y 163.822,Z 375.819,A -85,B 0,C 180,E1 -25696.832,E2 -25696.832} C_VEL
LIN {X 0,Y 154.155,Z 374.836,A -85,B 0,C 180,E1 -25700.337,E2 -25700.337} C_VEL
LIN {X 0,Y 145.177,Z 372.82,A -85,B 0,C 180,E1 -25704.485,E2 -25704.485} C_VEL
LIN {X 0,Y 137.54,Z 369.794,A -85,B 0,C 180,E1 -25709.271,E2 -25709.271} C_VEL
LIN {X 0,Y 131.188,Z 365.695,A -85,B 0,C 180,E1 -25714.623,E2 -25714.623} C_VEL
LIN {X 0,Y 127.068,Z 361.405,A -85,B 0,C 180,E1 -25719.49,E2 -25719.49} C_VEL
LIN {X 0,Y 124.86,Z 358.995,A -85,B 0,C 180,E1 -25721.721,E2 -25721.721} C_VEL
LIN {X 0,Y 120.418,Z 354.29,A -85,B 0,C 180,E1 -25725.219,E2 -25725.219} C_VEL
LIN {X 0,Y 116.639,Z 349.001,A -85,B 0,C 180,E1 -25728.859,E2 -25728.859} C_VEL
LIN {X 0,Y 115.547,Z 345.764,A -85,B 0,C 180,E1 -25731.256,E2 -25731.256} C_VEL
LIN {X 0,Y 114.947,Z 337.174,A -85,B 0,C 180,E1 -25737.372,E2 -25737.372} C_VEL
LIN {X 0,Y 114.968,Z 328.119,A -85,B 0,C 180,E1 -25742.628,E2 -25742.628} C_VEL
LIN {X 0,Y 115.452,Z 317.074,A -85,B 0,C 180,E1 -25747.873,E2 -25747.873} C_VEL
LIN {X 0,Y 116.216,Z 306.121,A -85,B 0,C 180,E1 -25752.114,E2 -25752.114} C_VEL
LIN {X 0,Y 117.314,Z 294.121,A -85,B 0,C 180,E1 -25755.869,E2 -25755.869} C_VEL
LIN {X 0,Y 118.097,Z 285.481,A -85,B 0,C 180,E1 -25758.115,E2 -25758.115} C_VEL
LIN {X 0,Y 116.113,Z 271.749,A -85,B 0,C 180,E1 -25760.784,E2 -25760.784} C_VEL
LIN {X 0,Y 115.086,Z 260.955,A -85,B 0,C 180,E1 -25762.493,E2 -25762.493} C_VEL
LIN {X 0,Y 116.295,Z 248.761,A -85,B 0,C 180,E1 -25772.949,E2 -25772.949} C_VEL
LIN {X 0,Y 116.669,Z 246.451,A -85,B 0,C 180,E1 -25774.909,E2 -25774.909} C_VEL
LIN {X 0,Y 117.284,Z 248.062,A -85,B 0,C 180,E1 -25775.75,E2 -25775.75} C_VEL
LIN {X 0,Y 118.972,Z 248.862,A -85,B 0,C 180,E1 -25777.197,E2 -25777.197} C_VEL
LIN {X 0,Y 121.249,Z 249.044,A -85,B 0,C 180,E1 -25778.834,E2 -25778.834} C_VEL
LIN {X 0,Y 122.087,Z 249.906,A -85,B 0,C 180,E1 -25779.555,E2 -25779.555} C_VEL
LIN {X 0,Y 125.082,Z 254.423,A -85,B 0,C 180,E1 -25782.396,E2 -25782.396} C_VEL
LIN {X 0,Y 128.952,Z 262.264,A -85,B 0,C 180,E1 -25786.504,E2 -25786.504} C_VEL
LIN {X 0,Y 131.451,Z 268.686,A -85,B 0,C 180,E1 -25789.63,E2 -25789.63} C_VEL
LIN {X 0,Y 132.862,Z 275.157,A -85,B 0,C 180,E1 -25792.51,E2 -25792.51} C_VEL
LIN {X 0,Y 133.351,Z 281.93,A -85,B 0,C 180,E1 -25795.486,E2 -25795.486} C_VEL
LIN {X 0,Y 133.162,Z 287.602,A -85,B 0,C 180,E1 -25798.14,E2 -25798.14} C_VEL
LIN {X 0,Y 131.771,Z 291.261,A -85,B 0,C 180,E1 -25799.692,E2 -25799.692} C_VEL
LIN {X 0,Y 128.82,Z 297.185,A -85,B 0,C 180,E1 -25802.368,E2 -25802.368} C_VEL
LIN {X 0,Y 125.183,Z 303.293,A -85,B 0,C 180,E1 -25805.977,E2 -25805.977} C_VEL
LIN {X 0,Y 122.259,Z 308.064,A -85,B 0,C 180,E1 -25809.82,E2 -25809.82} C_VEL
LIN {X 0,Y 119.908,Z 312.23,A -85,B 0,C 180,E1 -25814.703,E2 -25814.703} C_VEL
LIN {X 0,Y 117.706,Z 315.169,A -85,B 0,C 180,E1 -25819.677,E2 -25819.677} C_VEL
LIN {X 0,Y 116.906,Z 316.393,A -85,B 0,C 180,E1 -25823.09,E2 -25823.09} C_VEL
LIN {X 0,Y 116.322,Z 317.146,A -85,B 0,C 180,E1 -25826.532,E2 -25826.532} C_VEL
LIN {X 0,Y 116.112,Z 317.422,A -85,B 0,C 180,E1 -25829.996,E2 -25829.996} C_VEL
LIN {X 0,Y 116.321,Z 317.177,A -85,B 0,C 180,E1 -25833.459,E2 -25833.459} C_VEL
LIN {X 0,Y 116.903,Z 316.465,A -85,B 0,C 180,E1 -25836.901,E2 -25836.901} C_VEL
LIN {X 0,Y 117.703,Z 315.263,A -85,B 0,C 180,E1 -25840.314,E2 -25840.314} C_VEL
LIN {X 0,Y 119.89,Z 312.389,A -85,B 0,C 180,E1 -25845.29,E2 -25845.29} C_VEL
LIN {X 0,Y 122.21,Z 308.286,A -85,B 0,C 180,E1 -25850.18,E2 -25850.18} C_VEL
LIN {X 0,Y 123.55,Z 306.514,A -85,B 0,C 180,E1 -25851.695,E2 -25851.695} C_VEL
LIN {X 0,Y 125.851,Z 302.487,A -85,B 0,C 180,E1 -25854.756,E2 -25854.756} C_VEL
LIN {X 0,Y 129.551,Z 296.069,A -85,B 0,C 180,E1 -25858.334,E2 -25858.334} C_VEL
LIN {X 0,Y 132.558,Z 289.852,A -85,B 0,C 180,E1 -25861.077,E2 -25861.077} C_VEL
LIN {X 0,Y 133.228,Z 288.08,A -85,B 0,C 180,E1 -25861.833,E2 -25861.833} C_VEL
LIN {X 0,Y 133.381,Z 280.319,A -85,B 0,C 180,E1 -25865.418,E2 -25865.418} C_VEL
LIN {X 0,Y 132.814,Z 274.175,A -85,B 0,C 180,E1 -25868.12,E2 -25868.12} C_VEL
LIN {X 0,Y 131.617,Z 268.995,A -85,B 0,C 180,E1 -25870.455,E2 -25870.455} C_VEL
LIN {X 0,Y 129.493,Z 263.375,A -85,B 0,C 180,E1 -25873.184,E2 -25873.184} C_VEL
LIN {X 0,Y 126.082,Z 256.404,A -85,B 0,C 180,E1 -25876.85,E2 -25876.85} C_VEL
LIN {X 0,Y 123.874,Z 252.772,A -85,B 0,C 180,E1 -25879.004,E2 -25879.004} C_VEL
LIN {X 0,Y 121.504,Z 248.896,A -85,B 0,C 180,E1 -25881.352,E2 -25881.352} C_VEL
LIN {X 0,Y 119.049,Z 246.007,A -85,B 0,C 180,E1 -25883.662,E2 -25883.662} C_VEL
LIN {X 0,Y 118.288,Z 244.243,A -85,B 0,C 180,E1 -25884.65,E2 -25884.65} C_VEL
LIN {X 0,Y 118.228,Z 243.502,A -85,B 0,C 180,E1 -25887.656,E2 -25887.656} C_VEL
LIN {X 0,Y 118.122,Z 242.469,A -85,B 0,C 180,E1 -25893.174,E2 -25893.174} C_VEL
LIN {X 0,Y 118.064,Z 241.751,A -85,B 0,C 180,E1 -25899.074,E2 -25899.074} C_VEL
LIN {X 0,Y 118.093,Z 241.45,A -85,B 0,C 180,E1 -25902.688,E2 -25902.688} C_VEL
LIN {X 0,Y 118.418,Z 241.316,A -85,B 0,C 180,E1 -25909.744,E2 -25909.744} C_VEL
LIN {X 0,Y 118.895,Z 241.81,A -85,B 0,C 180,E1 -25916.611,E2 -25916.611} C_VEL
LIN {X 0,Y 119.286,Z 242.253,A -85,B 0,C 180,E1 -25920,E2 -25920} C_VEL
LIN {X 0,Y 119.197,Z 243.985,A -85,B 0,C 180,E1 -25926.772,E2 -25926.772} C_VEL
LIN {X 0,Y 119.351,Z 245.046,A -85,B 0,C 180,E1 -25930.175,E2 -25930.175} C_VEL
LIN {X 0,Y 119.445,Z 246.325,A -85,B 0,C 180,E1 -25933.612,E2 -25933.612} C_VEL
LIN {X 0,Y 119.83,Z 249.375,A -85,B 0,C 180,E1 -25940.603,E2 -25940.603} C_VEL
LIN {X 0,Y 120.786,Z 253.072,A -85,B 0,C 180,E1 -25947.741,E2 -25947.741} C_VEL
LIN {X 0,Y 121.419,Z 255.878,A -85,B 0,C 180,E1 -25952.372,E2 -25952.372} C_VEL
LIN {X 0,Y 123.252,Z 259.948,A -85,B 0,C 180,E1 -25954.146,E2 -25954.146} C_VEL
LIN {X 0,Y 124.889,Z 262.468,A -85,B 0,C 180,E1 -25955.516,E2 -25955.516} C_VEL
LIN {X 0,Y 127.01,Z 267.141,A -85,B 0,C 180,E1 -25957.494,E2 -25957.494} C_VEL
LIN {X 0,Y 130.858,Z 276.505,A -85,B 0,C 180,E1 -25961.252,E2 -25961.252} C_VEL
LIN {X 0,Y 132.829,Z 282.328,A -85,B 0,C 180,E1 -25963.459,E2 -25963.459} C_VEL
LIN {X 0,Y 133.032,Z 283.731,A -85,B 0,C 180,E1 -25963.898,E2 -25963.898} C_VEL
LIN {X 0,Y 131.438,Z 294.588,A -85,B 0,C 180,E1 -25966.5,E2 -25966.5} C_VEL
LIN {X 0,Y 129.003,Z 305.397,A -85,B 0,C 180,E1 -25969.704,E2 -25969.704} C_VEL
LIN {X 0,Y 126.055,Z 314.919,A -85,B 0,C 180,E1 -25973.182,E2 -25973.182} C_VEL
LIN {X 0,Y 123.689,Z 321.866,A -85,B 0,C 180,E1 -25976.364,E2 -25976.364} C_VEL
LIN {X 0,Y 121.446,Z 328.176,A -85,B 0,C 180,E1 -25979.892,E2 -25979.892} C_VEL
LIN {X 0,Y 118.206,Z 334.785,A -85,B 0,C 180,E1 -25984.471,E2 -25984.471} C_VEL
LIN {X 0,Y 116.11,Z 339.432,A -85,B 0,C 180,E1 -25988.71,E2 -25988.71} C_VEL
LIN {X 0,Y 114.608,Z 343.75,A -85,B 0,C 180,E1 -25993.986,E2 -25993.986} C_VEL
LIN {X 0,Y 114.21,Z 347.113,A -85,B 0,C 180,E1 -25999.924,E2 -25999.924} C_VEL
LIN {X 0,Y 114.583,Z 348.304,A -85,B 0,C 180,E1 -26002.958,E2 -26002.958} C_VEL
LIN {X 0,Y 115.394,Z 349.222,A -85,B 0,C 180,E1 -26006.513,E2 -26006.513} C_VEL
LIN {X 0,Y 117.381,Z 349.698,A -85,B 0,C 180,E1 -26011.72,E2 -26011.72} C_VEL
LIN {X 0,Y 118.039,Z 349.821,A -85,B 0,C 180,E1 -26013.204,E2 -26013.204} C_VEL
LIN {X 0,Y 117.87,Z 352.159,A -85,B 0,C 180,E1 -26015.136,E2 -26015.136} C_VEL
LIN {X 0,Y 117.077,Z 358.77,A -85,B 0,C 180,E1 -26022.133,E2 -26022.133} C_VEL
LIN {X 0,Y 118.161,Z 363.997,A -85,B 0,C 180,E1 -26029.099,E2 -26029.099} C_VEL
LIN {X 0,Y 120.315,Z 367.187,A -85,B 0,C 180,E1 -26034.14,E2 -26034.14} C_VEL
LIN {X 0,Y 125.045,Z 370.607,A -85,B 0,C 180,E1 -26040.391,E2 -26040.391} C_VEL
LIN {X 0,Y 131.452,Z 373.077,A -85,B 0,C 180,E1 -26046.027,E2 -26046.027} C_VEL
LIN {X 0,Y 139.295,Z 374.651,A -85,B 0,C 180,E1 -26050.993,E2 -26050.993} C_VEL
LIN {X 0,Y 148.616,Z 375.448,A -85,B 0,C 180,E1 -26055.186,E2 -26055.186} C_VEL
LIN {X 0,Y 150.873,Z 375.539,A -85,B 0,C 180,E1 -26056.033,E2 -26056.033} C_VEL
LIN {X 0,Y 152.153,Z 375.369,A -85,B 0,C 180,E1 -26057.315,E2 -26057.315} C_VEL
LIN {X 0,Y 143.997,Z 373.657,A -85,B 0,C 180,E1 -26060.618,E2 -26060.618} C_VEL
LIN {X 0,Y 135.317,Z 370.714,A -85,B 0,C 180,E1 -26065.158,E2 -26065.158} C_VEL
LIN {X 0,Y 127.997,Z 366.762,A -85,B 0,C 180,E1 -26070.385,E2 -26070.385} C_VEL
LIN {X 0,Y 122.284,Z 361.738,A -85,B 0,C 180,E1 -26076.277,E2 -26076.277} C_VEL
LIN {X 0,Y 118.913,Z 357.155,A -85,B 0,C 180,E1 -26081.033,E2 -26081.033} C_VEL
LIN {X 0,Y 116.27,Z 349.945,A -85,B 0,C 180,E1 -26087.786,E2 -26087.786} C_VEL
LIN {X 0,Y 115.547,Z 345.764,A -85,B 0,C 180,E1 -26091.256,E2 -26091.256} C_VEL
LIN {X 0,Y 114.59,Z 342.373,A -85,B 0,C 180,E1 -26093.596,E2 -26093.596} C_VEL
LIN {X 0,Y 112.917,Z 338.591,A -85,B 0,C 180,E1 -26095.738,E2 -26095.738} C_VEL
LIN {X 0,Y 109.314,Z 330.334,A -85,B 0,C 180,E1 -26099.845,E2 -26099.845} C_VEL
LIN {X 0,Y 108.38,Z 326.016,A -85,B 0,C 180,E1 -26102.003,E2 -26102.003} C_VEL
LIN {X 0,Y 108.332,Z 324.567,A -85,B 0,C 180,E1 -26102.751,E2 -26102.751} C_VEL
LIN {X 0,Y 108.861,Z 312.75,A -85,B 0,C 180,E1 -26108.352,E2 -26108.352} C_VEL
LIN {X 0,Y 109.733,Z 300.556,A -85,B 0,C 180,E1 -26112.954,E2 -26112.954} C_VEL
LIN {X 0,Y 110.899,Z 287.877,A -85,B 0,C 180,E1 -26116.808,E2 -26116.808} C_VEL
LIN {X 0,Y 111.091,Z 285.276,A -85,B 0,C 180,E1 -26117.474,E2 -26117.474} C_VEL
LIN {X 0,Y 109.053,Z 271.562,A -85,B 0,C 180,E1 -26120.267,E2 -26120.267} C_VEL
LIN {X 0,Y 108.054,Z 261.209,A -85,B 0,C 180,E1 -26122.088,E2 -26122.088} C_VEL
LIN {X 0,Y 108.441,Z 253.751,A -85,B 0,C 180,E1 -26128.95,E2 -26128.95} C_VEL
LIN {X 0,Y 108.958,Z 255.1,A -85,B 0,C 180,E1 -26129.993,E2 -26129.993} C_VEL
LIN {X 0,Y 109.634,Z 255.53,A -85,B 0,C 180,E1 -26130.853,E2 -26130.853} C_VEL
LIN {X 0,Y 111.616,Z 255.474,A -85,B 0,C 180,E1 -26132.793,E2 -26132.793} C_VEL
LIN {X 0,Y 113.111,Z 254.958,A -85,B 0,C 180,E1 -26134.001,E2 -26134.001} C_VEL
LIN {X 0,Y 118.536,Z 255.697,A -85,B 0,C 180,E1 -26138.502,E2 -26138.502} C_VEL
LIN {X 0,Y 121.967,Z 261.76,A -85,B 0,C 180,E1 -26142.503,E2 -26142.503} C_VEL
LIN {X 0,Y 125.174,Z 269.505,A -85,B 0,C 180,E1 -26146.878,E2 -26146.878} C_VEL
LIN {X 0,Y 126.842,Z 276.103,A -85,B 0,C 180,E1 -26150.244,E2 -26150.244} C_VEL
LIN {X 0,Y 127.338,Z 283.104,A -85,B 0,C 180,E1 -26153.604,E2 -26153.604} C_VEL
LIN {X 0,Y 127.066,Z 288.718,A -85,B 0,C 180,E1 -26156.416,E2 -26156.416} C_VEL
LIN {X 0,Y 126.296,Z 291.228,A -85,B 0,C 180,E1 -26157.621,E2 -26157.621} C_VEL
LIN {X 0,Y 122.643,Z 298.202,A -85,B 0,C 180,E1 -26160.846,E2 -26160.846} C_VEL
LIN {X 0,Y 118.798,Z 304.294,A -85,B 0,C 180,E1 -26164.597,E2 -26164.597} C_VEL
LIN {X 0,Y 115.686,Z 309.051,A -85,B 0,C 180,E1 -26168.618,E2 -26168.618} C_VEL
LIN {X 0,Y 113.143,Z 313.208,A -85,B 0,C 180,E1 -26173.764,E2 -26173.764} C_VEL
LIN {X 0,Y 110.799,Z 316.143,A -85,B 0,C 180,E1 -26179.026,E2 -26179.026} C_VEL
LIN {X 0,Y 109.932,Z 317.368,A -85,B 0,C 180,E1 -26182.649,E2 -26182.649} C_VEL
LIN {X 0,Y 109.308,Z 318.12,A -85,B 0,C 180,E1 -26186.309,E2 -26186.309} C_VEL
LIN {X 0,Y 109.084,Z 318.396,A -85,B 0,C 180,E1 -26189.995,E2 -26189.995} C_VEL
LIN {X 0,Y 109.307,Z 318.15,A -85,B 0,C 180,E1 -26193.682,E2 -26193.682} C_VEL
LIN {X 0,Y 109.929,Z 317.439,A -85,B 0,C 180,E1 -26197.341,E2 -26197.341} C_VEL
LIN {X 0,Y 110.796,Z 316.235,A -85,B 0,C 180,E1 -26200.965,E2 -26200.965} C_VEL
LIN {X 0,Y 113.126,Z 313.366,A -85,B 0,C 180,E1 -26206.229,E2 -26206.229} C_VEL
LIN {X 0,Y 115.637,Z 309.269,A -85,B 0,C 180,E1 -26211.382,E2 -26211.382} C_VEL
LIN {X 0,Y 117.048,Z 307.498,A -85,B 0,C 180,E1 -26212.967,E2 -26212.967} C_VEL
LIN {X 0,Y 119.507,Z 303.483,A -85,B 0,C 180,E1 -26216.167,E2 -26216.167} C_VEL
LIN {X 0,Y 123.416,Z 297.086,A -85,B 0,C 180,E1 -26219.881,E2 -26219.881} C_VEL
LIN {X 0,Y 126.862,Z 290.272,A -85,B 0,C 180,E1 -26222.999,E2 -26222.999} C_VEL
LIN {X 0,Y 127.359,Z 285.481,A -85,B 0,C 180,E1 -26225.402,E2 -26225.402} C_VEL
LIN {X 0,Y 127.309,Z 280.21,A -85,B 0,C 180,E1 -26227.978,E2 -26227.978} C_VEL
LIN {X 0,Y 126.82,Z 275.292,A -85,B 0,C 180,E1 -26230.361,E2 -26230.361} C_VEL
LIN {X 0,Y 125.352,Z 269.795,A -85,B 0,C 180,E1 -26233.209,E2 -26233.209} C_VEL
LIN {X 0,Y 122.405,Z 262.636,A -85,B 0,C 180,E1 -26237.273,E2 -26237.273} C_VEL
LIN {X 0,Y 118.099,Z 254.786,A -85,B 0,C 180,E1 -26242.412,E2 -26242.412} C_VEL
LIN {X 0,Y 115.733,Z 251.558,A -85,B 0,C 180,E1 -26245.089,E2 -26245.089} C_VEL
LIN {X 0,Y 114.945,Z 250.191,A -85,B 0,C 180,E1 -26246.073,E2 -26246.073} C_VEL
LIN {X 0,Y 112.161,Z 247.072,A -85,B 0,C 180,E1 -26249.395,E2 -26249.395} C_VEL
LIN {X 0,Y 111.426,Z 245.425,A -85,B 0,C 180,E1 -26250.681,E2 -26250.681} C_VEL
LIN {X 0,Y 111.469,Z 244.901,A -85,B 0,C 180,E1 -26253.81,E2 -26253.81} C_VEL
LIN {X 0,Y 111.426,Z 244.467,A -85,B 0,C 180,E1 -26257.763,E2 -26257.763} C_VEL
LIN {X 0,Y 111.468,Z 244.206,A -85,B 0,C 180,E1 -26261.624,E2 -26261.624} C_VEL
LIN {X 0,Y 111.584,Z 244.03,A -85,B 0,C 180,E1 -26265.408,E2 -26265.408} C_VEL
LIN {X 0,Y 111.78,Z 243.999,A -85,B 0,C 180,E1 -26269.127,E2 -26269.127} C_VEL
LIN {X 0,Y 112.295,Z 244.479,A -85,B 0,C 180,E1 -26276.412,E2 -26276.412} C_VEL
LIN {X 0,Y 112.716,Z 244.957,A -85,B 0,C 180,E1 -26280,E2 -26280} C_VEL
LIN {X 0,Y 112.632,Z 246.793,A -85,B 0,C 180,E1 -26287.169,E2 -26287.169} C_VEL
LIN {X 0,Y 112.741,Z 247.908,A -85,B 0,C 180,E1 -26290.778,E2 -26290.778} C_VEL
LIN {X 0,Y 112.987,Z 250.721,A -85,B 0,C 180,E1 -26298.12,E2 -26298.12} C_VEL
LIN {X 0,Y 113.785,Z 254.583,A -85,B 0,C 180,E1 -26306.356,E2 -26306.356} C_VEL
LIN {X 0,Y 116.463,Z 259.705,A -85,B 0,C 180,E1 -26309.563,E2 -26309.563} C_VEL
LIN {X 0,Y 117.976,Z 261.776,A -85,B 0,C 180,E1 -26311.09,E2 -26311.09} C_VEL
LIN {X 0,Y 119.954,Z 266.132,A -85,B 0,C 180,E1 -26313.317,E2 -26313.317} C_VEL
LIN {X 0,Y 120.957,Z 268.113,A -85,B 0,C 180,E1 -26314.381,E2 -26314.381} C_VEL
LIN {X 0,Y 124.457,Z 276.764,A -85,B 0,C 180,E1 -26318.401,E2 -26318.401} C_VEL
LIN {X 0,Y 127.268,Z 285.632,A -85,B 0,C 180,E1 -26322.15,E2 -26322.15} C_VEL
LIN {X 0,Y 125.736,Z 294.78,A -85,B 0,C 180,E1 -26324.555,E2 -26324.555} C_VEL
LIN {X 0,Y 122.963,Z 305.773,A -85,B 0,C 180,E1 -26327.989,E2 -26327.989} C_VEL
LIN {X 0,Y 120.246,Z 313.821,A -85,B 0,C 180,E1 -26331.081,E2 -26331.081} C_VEL
LIN {X 0,Y 117.048,Z 322.303,A -85,B 0,C 180,E1 -26335.226,E2 -26335.226} C_VEL
LIN {X 0,Y 114.704,Z 328.28,A -85,B 0,C 180,E1 -26338.825,E2 -26338.825} C_VEL
LIN {X 0,Y 111.767,Z 333.769,A -85,B 0,C 180,E1 -26342.883,E2 -26342.883} C_VEL
LIN {X 0,Y 109.451,Z 338.426,A -85,B 0,C 180,E1 -26347.345,E2 -26347.345} C_VEL
LIN {X 0,Y 107.694,Z 342.748,A -85,B 0,C 180,E1 -26352.928,E2 -26352.928} C_VEL
LIN {X 0,Y 107.14,Z 346.318,A -85,B 0,C 180,E1 -26359.721,E2 -26359.721} C_VEL
LIN {X 0,Y 108.204,Z 348.224,A -85,B 0,C 180,E1 -26366.281,E2 -26366.281} C_VEL
LIN {X 0,Y 109.487,Z 348.692,A -85,B 0,C 180,E1 -26370.005,E2 -26370.005} C_VEL
LIN {X 0,Y 111.576,Z 348.483,A -85,B 0,C 180,E1 -26375.086,E2 -26375.086} C_VEL
LIN {X 0,Y 110.777,Z 354.251,A -85,B 0,C 180,E1 -26380.977,E2 -26380.977} C_VEL
LIN {X 0,Y 111.494,Z 360.094,A -85,B 0,C 180,E1 -26388.376,E2 -26388.376} C_VEL
LIN {X 0,Y 114.28,Z 364.755,A -85,B 0,C 180,E1 -26395.503,E2 -26395.503} C_VEL
LIN {X 0,Y 119.262,Z 368.497,A -85,B 0,C 180,E1 -26402.035,E2 -26402.035} C_VEL
LIN {X 0,Y 125.955,Z 371.295,A -85,B 0,C 180,E1 -26407.868,E2 -26407.868} C_VEL
LIN {X 0,Y 134.139,Z 373.227,A -85,B 0,C 180,E1 -26412.936,E2 -26412.936} C_VEL
LIN {X 0,Y 140.844,Z 374.148,A -85,B 0,C 180,E1 -26416.035,E2 -26416.035} C_VEL
LIN {X 0,Y 141.956,Z 374.068,A -85,B 0,C 180,E1 -26417.345,E2 -26417.345} C_VEL
LIN {X 0,Y 133.928,Z 371.579,A -85,B 0,C 180,E1 -26420.971,E2 -26420.971} C_VEL
LIN {X 0,Y 123.769,Z 366.638,A -85,B 0,C 180,E1 -26427.354,E2 -26427.354} C_VEL
LIN {X 0,Y 117.36,Z 361.505,A -85,B 0,C 180,E1 -26433.312,E2 -26433.312} C_VEL
LIN {X 0,Y 112.485,Z 355.151,A -85,B 0,C 180,E1 -26439.903,E2 -26439.903} C_VEL
LIN {X 0,Y 109.712,Z 347.542,A -85,B 0,C 180,E1 -26447.044,E2 -26447.044} C_VEL
LIN {X 0,Y 108.673,Z 340.715,A -85,B 0,C 180,E1 -26452.569,E2 -26452.569} C_VEL
LIN {X 0,Y 108.331,Z 332.594,A -85,B 0,C 180,E1 -26458.141,E2 -26458.141} C_VEL
LIN {X 0,Y 108.332,Z 324.567,A -85,B 0,C 180,E1 -26462.751,E2 -26462.751} C_VEL
LIN {X 0,Y 107.833,Z 320.195,A -85,B 0,C 180,E1 -26464.816,E2 -26464.816} C_VEL
LIN {X 0,Y 106.52,Z 315.542,A -85,B 0,C 180,E1 -26466.645,E2 -26466.645} C_VEL
LIN {X 0,Y 103.181,Z 304.002,A -85,B 0,C 180,E1 -26470.59,E2 -26470.59} C_VEL
LIN {X 0,Y 102.934,Z 298.905,A -85,B 0,C 180,E1 -26472.355,E2 -26472.355} C_VEL
LIN {X 0,Y 104.036,Z 286.319,A -85,B 0,C 180,E1 -26476.331,E2 -26476.331} C_VEL
LIN {X 0,Y 103.895,Z 283.659,A -85,B 0,C 180,E1 -26477.011,E2 -26477.011} C_VEL
LIN {X 0,Y 101.885,Z 269.949,A -85,B 0,C 180,E1 -26479.868,E2 -26479.868} C_VEL
LIN {X 0,Y 101.066,Z 261.605,A -85,B 0,C 180,E1 -26481.413,E2 -26481.413} C_VEL
LIN {X 0,Y 100.972,Z 261.201,A -85,B 0,C 180,E1 -26481.836,E2 -26481.836} C_VEL
LIN {X 0,Y 101.021,Z 262.119,A -85,B 0,C 180,E1 -26482.497,E2 -26482.497} C_VEL
LIN {X 0,Y 101.887,Z 262.971,A -85,B 0,C 180,E1 -26484.448,E2 -26484.448} C_VEL
LIN {X 0,Y 104.804,Z 262.014,A -85,B 0,C 180,E1 -26487.996,E2 -26487.996} C_VEL
LIN {X 0,Y 107.707,Z 262.27,A -85,B 0,C 180,E1 -26491.468,E2 -26491.468} C_VEL
LIN {X 0,Y 111.738,Z 261.828,A -85,B 0,C 180,E1 -26495.141,E2 -26495.141} C_VEL
LIN {X 0,Y 114.745,Z 262.299,A -85,B 0,C 180,E1 -26497.77,E2 -26497.77} C_VEL
LIN {X 0,Y 116.184,Z 263.97,A -85,B 0,C 180,E1 -26499.431,E2 -26499.431} C_VEL
LIN {X 0,Y 118.491,Z 269.312,A -85,B 0,C 180,E1 -26503.008,E2 -26503.008} C_VEL
LIN {X 0,Y 120.496,Z 275.502,A -85,B 0,C 180,E1 -26506.807,E2 -26506.807} C_VEL
LIN {X 0,Y 121.314,Z 280.741,A -85,B 0,C 180,E1 -26509.707,E2 -26509.707} C_VEL
LIN {X 0,Y 121.276,Z 287.169,A -85,B 0,C 180,E1 -26513.097,E2 -26513.097} C_VEL
LIN {X 0,Y 120.784,Z 291.45,A -85,B 0,C 180,E1 -26515.438,E2 -26515.438} C_VEL
LIN {X 0,Y 117.42,Z 297.814,A -85,B 0,C 180,E1 -26518.413,E2 -26518.413} C_VEL
LIN {X 0,Y 113.256,Z 304.201,A -85,B 0,C 180,E1 -26522.259,E2 -26522.259} C_VEL
LIN {X 0,Y 109.17,Z 310.039,A -85,B 0,C 180,E1 -26527.273,E2 -26527.273} C_VEL
LIN {X 0,Y 106.413,Z 314.188,A -85,B 0,C 180,E1 -26532.706,E2 -26532.706} C_VEL
LIN {X 0,Y 103.909,Z 317.117,A -85,B 0,C 180,E1 -26538.288,E2 -26538.288} C_VEL
LIN {X 0,Y 102.966,Z 318.343,A -85,B 0,C 180,E1 -26542.149,E2 -26542.149} C_VEL
LIN {X 0,Y 102.296,Z 319.094,A -85,B 0,C 180,E1 -26546.055,E2 -26546.055} C_VEL
LIN {X 0,Y 102.056,Z 319.37,A -85,B 0,C 180,E1 -26549.995,E2 -26549.995} C_VEL
LIN {X 0,Y 102.294,Z 319.123,A -85,B 0,C 180,E1 -26553.934,E2 -26553.934} C_VEL
LIN {X 0,Y 102.963,Z 318.413,A -85,B 0,C 180,E1 -26557.841,E2 -26557.841} C_VEL
LIN {X 0,Y 103.905,Z 317.208,A -85,B 0,C 180,E1 -26561.702,E2 -26561.702} C_VEL
LIN {X 0,Y 106.395,Z 314.342,A -85,B 0,C 180,E1 -26567.287,E2 -26567.287} C_VEL
LIN {X 0,Y 109.12,Z 310.251,A -85,B 0,C 180,E1 -26572.728,E2 -26572.728} C_VEL
LIN {X 0,Y 110.61,Z 308.482,A -85,B 0,C 180,E1 -26574.388,E2 -26574.388} C_VEL
LIN {X 0,Y 113.243,Z 304.478,A -85,B 0,C 180,E1 -26577.734,E2 -26577.734} C_VEL
LIN {X 0,Y 117.381,Z 298.103,A -85,B 0,C 180,E1 -26581.588,E2 -26581.588} C_VEL
LIN {X 0,Y 120.837,Z 291.74,A -85,B 0,C 180,E1 -26584.617,E2 -26584.617} C_VEL
LIN {X 0,Y 121.451,Z 286.618,A -85,B 0,C 180,E1 -26587.408,E2 -26587.408} C_VEL
LIN {X 0,Y 121.455,Z 281.173,A -85,B 0,C 180,E1 -26590.296,E2 -26590.296} C_VEL
LIN {X 0,Y 120.659,Z 275.841,A -85,B 0,C 180,E1 -26593.276,E2 -26593.276} C_VEL
LIN {X 0,Y 118.56,Z 269.375,A -85,B 0,C 180,E1 -26597.245,E2 -26597.245} C_VEL
LIN {X 0,Y 116.364,Z 264.352,A -85,B 0,C 180,E1 -26600.641,E2 -26600.641} C_VEL
LIN {X 0,Y 114.047,Z 260.075,A -85,B 0,C 180,E1 -26603.948,E2 -26603.948} C_VEL
LIN {X 0,Y 110.844,Z 255.196,A -85,B 0,C 180,E1 -26608.46,E2 -26608.46} C_VEL
LIN {X 0,Y 108.937,Z 252.107,A -85,B 0,C 180,E1 -26611.504,E2 -26611.504} C_VEL
LIN {X 0,Y 105.566,Z 248.604,A -85,B 0,C 180,E1 -26617.105,E2 -26617.105} C_VEL
LIN {X 0,Y 104.768,Z 246.931,A -85,B 0,C 180,E1 -26619.097,E2 -26619.097} C_VEL
LIN {X 0,Y 104.925,Z 246.682,A -85,B 0,C 180,E1 -26624.459,E2 -26624.459} C_VEL
LIN {X 0,Y 105.148,Z 246.691,A -85,B 0,C 180,E1 -26628.432,E2 -26628.432} C_VEL
LIN {X 0,Y 105.686,Z 247.12,A -85,B 0,C 180,E1 -26636.187,E2 -26636.187} C_VEL
LIN {X 0,Y 106.11,Z 247.591,A -85,B 0,C 180,E1 -26640,E2 -26640} C_VEL
LIN {X 0,Y 105.993,Z 249.478,A -85,B 0,C 180,E1 -26647.62,E2 -26647.62} C_VEL
LIN {X 0,Y 106.053,Z 250.659,A -85,B 0,C 180,E1 -26651.467,E2 -26651.467} C_VEL
LIN {X 0,Y 106.347,Z 253.242,A -85,B 0,C 180,E1 -26658.17,E2 -26658.17} C_VEL
LIN {X 0,Y 107.927,Z 256.902,A -85,B 0,C 180,E1 -26661.111,E2 -26661.111} C_VEL
LIN {X 0,Y 110.946,Z 261.041,A -85,B 0,C 180,E1 -26665.314,E2 -26665.314} C_VEL
LIN {X 0,Y 113.495,Z 266.032,A -85,B 0,C 180,E1 -26668.806,E2 -26668.806} C_VEL
LIN {X 0,Y 114.302,Z 267.442,A -85,B 0,C 180,E1 -26669.798,E2 -26669.798} C_VEL
LIN {X 0,Y 117.139,Z 274.433,A -85,B 0,C 180,E1 -26673.709,E2 -26673.709} C_VEL
LIN {X 0,Y 119.539,Z 281.199,A -85,B 0,C 180,E1 -26677.18,E2 -26677.18} C_VEL
LIN {X 0,Y 121.56,Z 288.433,A -85,B 0,C 180,E1 -26680.573,E2 -26680.573} C_VEL
LIN {X 0,Y 119.455,Z 297.843,A -85,B 0,C 180,E1 -26683.296,E2 -26683.296} C_VEL
LIN {X 0,Y 116.623,Z 307.258,A -85,B 0,C 180,E1 -26686.589,E2 -26686.589} C_VEL
LIN {X 0,Y 113.853,Z 314.507,A -85,B 0,C 180,E1 -26689.604,E2 -26689.604} C_VEL
LIN {X 0,Y 111.07,Z 321.232,A -85,B 0,C 180,E1 -26693.056,E2 -26693.056} C_VEL
LIN {X 0,Y 108.604,Z 327.248,A -85,B 0,C 180,E1 -26696.857,E2 -26696.857} C_VEL
LIN {X 0,Y 104.844,Z 333.767,A -85,B 0,C 180,E1 -26702.022,E2 -26702.022} C_VEL
LIN {X 0,Y 102.047,Z 338.999,A -85,B 0,C 180,E1 -26707.747,E2 -26707.747} C_VEL
LIN {X 0,Y 100.463,Z 342.933,A -85,B 0,C 180,E1 -26713.756,E2 -26713.756} C_VEL
LIN {X 0,Y 100.078,Z 345.49,A -85,B 0,C 180,E1 -26719.467,E2 -26719.467} C_VEL
LIN {X 0,Y 101.011,Z 347.224,A -85,B 0,C 180,E1 -26726.016,E2 -26726.016} C_VEL
LIN {X 0,Y 102.304,Z 347.697,A -85,B 0,C 180,E1 -26730.005,E2 -26730.005} C_VEL
LIN {X 0,Y 103.925,Z 347.608,A -85,B 0,C 180,E1 -26733.883,E2 -26733.883} C_VEL
LIN {X 0,Y 105.061,Z 347.191,A -85,B 0,C 180,E1 -26737.452,E2 -26737.452} C_VEL
LIN {X 0,Y 104.771,Z 354.309,A -85,B 0,C 180,E1 -26745.569,E2 -26745.569} C_VEL
LIN {X 0,Y 107.35,Z 361.001,A -85,B 0,C 180,E1 -26755.19,E2 -26755.19} C_VEL
LIN {X 0,Y 113.64,Z 366.185,A -85,B 0,C 180,E1 -26763.826,E2 -26763.826} C_VEL
LIN {X 0,Y 120.647,Z 369.306,A -85,B 0,C 180,E1 -26769.855,E2 -26769.855} C_VEL
LIN {X 0,Y 131.08,Z 371.946,A -85,B 0,C 180,E1 -26775.96,E2 -26775.96} C_VEL
LIN {X 0,Y 132.068,Z 371.935,A -85,B 0,C 180,E1 -26777.355,E2 -26777.355} C_VEL
LIN {X 0,Y 121.979,Z 367.543,A -85,B 0,C 180,E1 -26782.773,E2 -26782.773} C_VEL
LIN {X 0,Y 114.395,Z 362.542,A -85,B 0,C 180,E1 -26788.52,E2 -26788.52} C_VEL
LIN {X 0,Y 108.339,Z 356.273,A -85,B 0,C 180,E1 -26795.266,E2 -26795.266} C_VEL
LIN {X 0,Y 104.132,Z 348.081,A -85,B 0,C 180,E1 -26803.331,E2 -26803.331} C_VEL
LIN {X 0,Y 102.483,Z 340.264,A -85,B 0,C 180,E1 -26810.128,E2 -26810.128} C_VEL
LIN {X 0,Y 101.808,Z 330.712,A -85,B 0,C 180,E1 -26817.032,E2 -26817.032} C_VEL
LIN {X 0,Y 101.728,Z 322.369,A -85,B 0,C 180,E1 -26821.98,E2 -26821.98} C_VEL
LIN {X 0,Y 102.134,Z 311.375,A -85,B 0,C 180,E1 -26827.413,E2 -26827.413} C_VEL
LIN {X 0,Y 102.934,Z 298.905,A -85,B 0,C 180,E1 -26832.355,E2 -26832.355} C_VEL
LIN {X 0,Y 102.584,Z 295.5,A -85,B 0,C 180,E1 -26833.417,E2 -26833.417} C_VEL
LIN {X 0,Y 101.336,Z 292.053,A -85,B 0,C 180,E1 -26834.281,E2 -26834.281} C_VEL
LIN {X 0,Y 97.001,Z 282.699,A -85,B 0,C 180,E1 -26836.261,E2 -26836.261} C_VEL
LIN {X 0,Y 96.402,Z 280.179,A -85,B 0,C 180,E1 -26836.824,E2 -26836.824} C_VEL
LIN {X 0,Y 95.136,Z 271.721,A -85,B 0,C 180,E1 -26838.67,E2 -26838.67} C_VEL
LIN {X 0,Y 95.086,Z 272.802,A -85,B 0,C 180,E1 -26839.83,E2 -26839.83} C_VEL
LIN {X 0,Y 95.883,Z 272.736,A -85,B 0,C 180,E1 -26841.499,E2 -26841.499} C_VEL
LIN {X 0,Y 96.737,Z 271.973,A -85,B 0,C 180,E1 -26842.422,E2 -26842.422} C_VEL
LIN {X 0,Y 97.815,Z 270.723,A -85,B 0,C 180,E1 -26843.277,E2 -26843.277} C_VEL
LIN {X 0,Y 99.458,Z 269.521,A -85,B 0,C 180,E1 -26845.086,E2 -26845.086} C_VEL
LIN {X 0,Y 102.443,Z 268.625,A -85,B 0,C 180,E1 -26848.701,E2 -26848.701} C_VEL
LIN {X 0,Y 105.404,Z 268.815,A -85,B 0,C 180,E1 -26852.237,E2 -26852.237} C_VEL
LIN {X 0,Y 108.978,Z 268.35,A -85,B 0,C 180,E1 -26855.48,E2 -26855.48} C_VEL
LIN {X 0,Y 112.158,Z 269.757,A -85,B 0,C 180,E1 -26858.801,E2 -26858.801} C_VEL
LIN {X 0,Y 113.991,Z 275.122,A -85,B 0,C 180,E1 -26862.703,E2 -26862.703} C_VEL
LIN {X 0,Y 115.291,Z 280.545,A -85,B 0,C 180,E1 -26866.293,E2 -26866.293} C_VEL
LIN {X 0,Y 115.65,Z 285.021,A -85,B 0,C 180,E1 -26868.94,E2 -26868.94} C_VEL
LIN {X 0,Y 115.197,Z 291.062,A -85,B 0,C 180,E1 -26872.478,E2 -26872.478} C_VEL
LIN {X 0,Y 114.799,Z 292.952,A -85,B 0,C 180,E1 -26873.644,E2 -26873.644} C_VEL
LIN {X 0,Y 111.5,Z 298.844,A -85,B 0,C 180,E1 -26876.523,E2 -26876.523} C_VEL
LIN {X 0,Y 107.087,Z 305.2,A -85,B 0,C 180,E1 -26880.509,E2 -26880.509} C_VEL
LIN {X 0,Y 102.721,Z 311.025,A -85,B 0,C 180,E1 -26885.758,E2 -26885.758} C_VEL
LIN {X 0,Y 99.724,Z 315.166,A -85,B 0,C 180,E1 -26891.505,E2 -26891.505} C_VEL
LIN {X 0,Y 97.038,Z 318.091,A -85,B 0,C 180,E1 -26897.446,E2 -26897.446} C_VEL
LIN {X 0,Y 96.009,Z 319.317,A -85,B 0,C 180,E1 -26901.576,E2 -26901.576} C_VEL
LIN {X 0,Y 95.286,Z 320.068,A -85,B 0,C 180,E1 -26905.765,E2 -26905.765} C_VEL
LIN {X 0,Y 95.028,Z 320.344,A -85,B 0,C 180,E1 -26909.995,E2 -26909.995} C_VEL
LIN {X 0,Y 95.284,Z 320.097,A -85,B 0,C 180,E1 -26914.224,E2 -26914.224} C_VEL
LIN {X 0,Y 96.006,Z 319.387,A -85,B 0,C 180,E1 -26918.413,E2 -26918.413} C_VEL
LIN {X 0,Y 97.033,Z 318.181,A -85,B 0,C 180,E1 -26922.544,E2 -26922.544} C_VEL
LIN {X 0,Y 99.706,Z 315.318,A -85,B 0,C 180,E1 -26928.488,E2 -26928.488} C_VEL
LIN {X 0,Y 102.671,Z 311.232,A -85,B 0,C 180,E1 -26934.244,E2 -26934.244} C_VEL
LIN {X 0,Y 104.248,Z 309.468,A -85,B 0,C 180,E1 -26935.984,E2 -26935.984} C_VEL
LIN {X 0,Y 107.074,Z 305.474,A -85,B 0,C 180,E1 -26939.484,E2 -26939.484} C_VEL
LIN {X 0,Y 111.462,Z 299.122,A -85,B 0,C 180,E1 -26943.479,E2 -26943.479} C_VEL
LIN {X 0,Y 114.873,Z 293.218,A -85,B 0,C 180,E1 -26946.418,E2 -26946.418} C_VEL
LIN {X 0,Y 115.607,Z 287.952,A -85,B 0,C 180,E1 -26949.548,E2 -26949.548} C_VEL
LIN {X 0,Y 115.705,Z 283.09,A -85,B 0,C 180,E1 -26952.401,E2 -26952.401} C_VEL
LIN {X 0,Y 115.028,Z 278.43,A -85,B 0,C 180,E1 -26955.361,E2 -26955.361} C_VEL
LIN {X 0,Y 112.839,Z 271.363,A -85,B 0,C 180,E1 -26960.326,E2 -26960.326} C_VEL
LIN {X 0,Y 110.239,Z 265.718,A -85,B 0,C 180,E1 -26964.986,E2 -26964.986} C_VEL
LIN {X 0,Y 108.16,Z 261.882,A -85,B 0,C 180,E1 -26968.679,E2 -26968.679} C_VEL
LIN {X 0,Y 106.166,Z 258.581,A -85,B 0,C 180,E1 -26972.394,E2 -26972.394} C_VEL
LIN {X 0,Y 103.194,Z 254.708,A -85,B 0,C 180,E1 -26978.572,E2 -26978.572} C_VEL
LIN {X 0,Y 102.701,Z 253.641,A -85,B 0,C 180,E1 -26979.991,E2 -26979.991} C_VEL
LIN {X 0,Y 99.354,Z 250.577,A -85,B 0,C 180,E1 -26993.909,E2 -26993.909} C_VEL
LIN {X 0,Y 99.322,Z 250.274,A -85,B 0,C 180,E1 -26995.942,E2 -26995.942} C_VEL
LIN {X 0,Y 99.529,Z 250.515,A -85,B 0,C 180,E1 -27000.506,E2 -27000.506} C_VEL
LIN {X 0,Y 101.386,Z 255.878,A -85,B 0,C 180,E1 -27010.737,E2 -27010.737} C_VEL
LIN {X 0,Y 103.907,Z 259.634,A -85,B 0,C 180,E1 -27016.832,E2 -27016.832} C_VEL
LIN {X 0,Y 105.775,Z 264.075,A -85,B 0,C 180,E1 -27020.924,E2 -27020.924} C_VEL
LIN {X 0,Y 107.736,Z 267.006,A -85,B 0,C 180,E1 -27024.052,E2 -27024.052} C_VEL
LIN {X 0,Y 110.415,Z 272.931,A -85,B 0,C 180,E1 -27028.514,E2 -27028.514} C_VEL
LIN {X 0,Y 112.455,Z 278.651,A -85,B 0,C 180,E1 -27032.078,E2 -27032.078} C_VEL
LIN {X 0,Y 114.382,Z 285.113,A -85,B 0,C 180,E1 -27035.714,E2 -27035.714} C_VEL
LIN {X 0,Y 115.668,Z 290.496,A -85,B 0,C 180,E1 -27038.535,E2 -27038.535} C_VEL
LIN {X 0,Y 115.712,Z 291.952,A -85,B 0,C 180,E1 -27039.142,E2 -27039.142} C_VEL
LIN {X 0,Y 112.614,Z 302.376,A -85,B 0,C 180,E1 -27042.52,E2 -27042.52} C_VEL
LIN {X 0,Y 109.219,Z 311.62,A -85,B 0,C 180,E1 -27046.239,E2 -27046.239} C_VEL
LIN {X 0,Y 105.275,Z 320.162,A -85,B 0,C 180,E1 -27050.646,E2 -27050.646} C_VEL
LIN {X 0,Y 102.055,Z 327.239,A -85,B 0,C 180,E1 -27055.386,E2 -27055.386} C_VEL
LIN {X 0,Y 98.559,Z 332.759,A -85,B 0,C 180,E1 -27060.062,E2 -27060.062} C_VEL
LIN {X 0,Y 95.416,Z 337.993,A -85,B 0,C 180,E1 -27066.108,E2 -27066.108} C_VEL
LIN {X 0,Y 93.564,Z 341.933,A -85,B 0,C 180,E1 -27072.521,E2 -27072.521} C_VEL
LIN {X 0,Y 93.021,Z 344.652,A -85,B 0,C 180,E1 -27079.169,E2 -27079.169} C_VEL
LIN {X 0,Y 93.828,Z 346.227,A -85,B 0,C 180,E1 -27085.71,E2 -27085.71} C_VEL
LIN {X 0,Y 95.097,Z 346.698,A -85,B 0,C 180,E1 -27090.005,E2 -27090.005} C_VEL
LIN {X 0,Y 96.809,Z 346.619,A -85,B 0,C 180,E1 -27094.168,E2 -27094.168} C_VEL
LIN {X 0,Y 98.68,Z 345.573,A -85,B 0,C 180,E1 -27100.002,E2 -27100.002} C_VEL
LIN {X 0,Y 98.953,Z 352.625,A -85,B 0,C 180,E1 -27108.644,E2 -27108.644} C_VEL
LIN {X 0,Y 101.526,Z 358.108,A -85,B 0,C 180,E1 -27116.744,E2 -27116.744} C_VEL
LIN {X 0,Y 108.194,Z 363.676,A -85,B 0,C 180,E1 -27125.781,E2 -27125.781} C_VEL
LIN {X 0,Y 115.554,Z 367.106,A -85,B 0,C 180,E1 -27131.997,E2 -27131.997} C_VEL
LIN {X 0,Y 123.368,Z 369.433,A -85,B 0,C 180,E1 -27136.873,E2 -27136.873} C_VEL
LIN {X 0,Y 112.373,Z 363.467,A -85,B 0,C 180,E1 -27143.548,E2 -27143.548} C_VEL
LIN {X 0,Y 104.324,Z 356.474,A -85,B 0,C 180,E1 -27151.146,E2 -27151.146} C_VEL
LIN {X 0,Y 99.995,Z 350.455,A -85,B 0,C 180,E1 -27157.26,E2 -27157.26} C_VEL
LIN {X 0,Y 96.937,Z 342.032,A -85,B 0,C 180,E1 -27165.3,E2 -27165.3} C_VEL
LIN {X 0,Y 95.708,Z 334.448,A -85,B 0,C 180,E1 -27171.555,E2 -27171.555} C_VEL
LIN {X 0,Y 95.328,Z 327.039,A -85,B 0,C 180,E1 -27176.83,E2 -27176.83} C_VEL
LIN {X 0,Y 95.19,Z 318.162,A -85,B 0,C 180,E1 -27182.116,E2 -27182.116} C_VEL
LIN {X 0,Y 95.508,Z 307.462,A -85,B 0,C 180,E1 -27187.399,E2 -27187.399} C_VEL
LIN {X 0,Y 96.394,Z 294.36,A -85,B 0,C 180,E1 -27192.635,E2 -27192.635} C_VEL
LIN {X 0,Y 97.187,Z 284.704,A -85,B 0,C 180,E1 -27195.735,E2 -27195.735} C_VEL
LIN {X 0,Y 96.402,Z 280.179,A -85,B 0,C 180,E1 -27196.824,E2 -27196.824} C_VEL
LIN {X 0,Y 96.124,Z 277.948,A -85,B 0,C 180,E1 -27197.738,E2 -27197.738} C_VEL
LIN {X 0,Y 96.06,Z 275.867,A -85,B 0,C 180,E1 -27199.559,E2 -27199.559} C_VEL
LIN {X 0,Y 96.486,Z 274.466,A -85,B 0,C 180,E1 -27202.316,E2 -27202.316} C_VEL
LIN {X 0,Y 97.207,Z 274.134,A -85,B 0,C 180,E1 -27204.599,E2 -27204.599} C_VEL
LIN {X 0,Y 101.701,Z 274.999,A -85,B 0,C 180,E1 -27212.009,E2 -27212.009} C_VEL
LIN {X 0,Y 103.758,Z 275.042,A -85,B 0,C 180,E1 -27214.266,E2 -27214.266} C_VEL
LIN {X 0,Y 106.246,Z 274.848,A -85,B 0,C 180,E1 -27216.537,E2 -27216.537} C_VEL
LIN {X 0,Y 108.005,Z 275.865,A -85,B 0,C 180,E1 -27218.654,E2 -27218.654} C_VEL
LIN {X 0,Y 109.25,Z 280.884,A -85,B 0,C 180,E1 -27222.512,E2 -27222.512} C_VEL
LIN {X 0,Y 109.938,Z 285.786,A -85,B 0,C 180,E1 -27225.987,E2 -27225.987} C_VEL
LIN {X 0,Y 109.613,Z 290.658,A -85,B 0,C 180,E1 -27229.142,E2 -27229.142} C_VEL
LIN {X 0,Y 108.918,Z 294.528,A -85,B 0,C 180,E1 -27231.701,E2 -27231.701} C_VEL
LIN {X 0,Y 105.715,Z 299.874,A -85,B 0,C 180,E1 -27234.424,E2 -27234.424} C_VEL
LIN {X 0,Y 101.031,Z 306.199,A -85,B 0,C 180,E1 -27238.546,E2 -27238.546} C_VEL
LIN {X 0,Y 96.354,Z 312.01,A -85,B 0,C 180,E1 -27244.041,E2 -27244.041} C_VEL
LIN {X 0,Y 93.085,Z 316.143,A -85,B 0,C 180,E1 -27250.132,E2 -27250.132} C_VEL
LIN {X 0,Y 90.191,Z 319.065,A -85,B 0,C 180,E1 -27256.475,E2 -27256.475} C_VEL
LIN {X 0,Y 89.062,Z 320.292,A -85,B 0,C 180,E1 -27260.914,E2 -27260.914} C_VEL
LIN {X 0,Y 88.279,Z 321.041,A -85,B 0,C 180,E1 -27265.428,E2 -27265.428} C_VEL
LIN {X 0,Y 88,Z 321.319,A -85,B 0,C 180,E1 -27269.994,E2 -27269.994} C_VEL
LIN {X 0,Y 88.277,Z 321.071,A -85,B 0,C 180,E1 -27274.56,E2 -27274.56} C_VEL
LIN {X 0,Y 89.059,Z 320.361,A -85,B 0,C 180,E1 -27279.075,E2 -27279.075} C_VEL
LIN {X 0,Y 90.186,Z 319.154,A -85,B 0,C 180,E1 -27283.514,E2 -27283.514} C_VEL
LIN {X 0,Y 93.066,Z 316.296,A -85,B 0,C 180,E1 -27289.86,E2 -27289.86} C_VEL
LIN {X 0,Y 96.303,Z 312.212,A -85,B 0,C 180,E1 -27295.962,E2 -27295.962} C_VEL
LIN {X 0,Y 97.978,Z 310.452,A -85,B 0,C 180,E1 -27297.785,E2 -27297.785} C_VEL
LIN {X 0,Y 101.017,Z 306.471,A -85,B 0,C 180,E1 -27301.446,E2 -27301.446} C_VEL
LIN {X 0,Y 105.677,Z 300.141,A -85,B 0,C 180,E1 -27305.579,E2 -27305.579} C_VEL
LIN {X 0,Y 108.991,Z 294.741,A -85,B 0,C 180,E1 -27308.404,E2 -27308.404} C_VEL
LIN {X 0,Y 109.884,Z 289.508,A -85,B 0,C 180,E1 -27311.794,E2 -27311.794} C_VEL
LIN {X 0,Y 110.056,Z 285.25,A -85,B 0,C 180,E1 -27314.616,E2 -27314.616} C_VEL
LIN {X 0,Y 109.146,Z 279.933,A -85,B 0,C 180,E1 -27318.533,E2 -27318.533} C_VEL
LIN {X 0,Y 107.741,Z 275.029,A -85,B 0,C 180,E1 -27322.502,E2 -27322.502} C_VEL
LIN {X 0,Y 106.336,Z 271.496,A -85,B 0,C 180,E1 -27325.766,E2 -27325.766} C_VEL
LIN {X 0,Y 104.584,Z 267.705,A -85,B 0,C 180,E1 -27329.735,E2 -27329.735} C_VEL
LIN {X 0,Y 102.925,Z 264.544,A -85,B 0,C 180,E1 -27333.649,E2 -27333.649} C_VEL
LIN {X 0,Y 100.629,Z 261.145,A -85,B 0,C 180,E1 -27339.561,E2 -27339.561} C_VEL
LIN {X 0,Y 98.821,Z 259.216,A -85,B 0,C 180,E1 -27345.586,E2 -27345.586} C_VEL
LIN {X 0,Y 97.782,Z 257.244,A -85,B 0,C 180,E1 -27355.878,E2 -27355.878} C_VEL
LIN {X 0,Y 97.947,Z 257.363,A -85,B 0,C 180,E1 -27359.743,E2 -27359.743} C_VEL
LIN {X 0,Y 98.997,Z 261.944,A -85,B 0,C 180,E1 -27368.934,E2 -27368.934} C_VEL
LIN {X 0,Y 100.653,Z 264.911,A -85,B 0,C 180,E1 -27374.145,E2 -27374.145} C_VEL
LIN {X 0,Y 102.771,Z 270.33,A -85,B 0,C 180,E1 -27379.994,E2 -27379.994} C_VEL
LIN {X 0,Y 103.907,Z 272.097,A -85,B 0,C 180,E1 -27382.155,E2 -27382.155} C_VEL
LIN {X 0,Y 106.405,Z 278.679,A -85,B 0,C 180,E1 -27387.539,E2 -27387.539} C_VEL
LIN {X 0,Y 108.441,Z 285.679,A -85,B 0,C 180,E1 -27392.213,E2 -27392.213} C_VEL
LIN {X 0,Y 109.88,Z 292.692,A -85,B 0,C 180,E1 -27396.391,E2 -27396.391} C_VEL
LIN {X 0,Y 110.013,Z 294.27,A -85,B 0,C 180,E1 -27397.214,E2 -27397.214} C_VEL
LIN {X 0,Y 106.582,Z 304.178,A -85,B 0,C 180,E1 -27400.723,E2 -27400.723} C_VEL
LIN {X 0,Y 103.132,Z 312.32,A -85,B 0,C 180,E1 -27404.321,E2 -27404.321} C_VEL
LIN {X 0,Y 99.694,Z 319.091,A -85,B 0,C 180,E1 -27407.963,E2 -27407.963} C_VEL
LIN {X 0,Y 96.094,Z 326.189,A -85,B 0,C 180,E1 -27412.895,E2 -27412.895} C_VEL
LIN {X 0,Y 92.396,Z 331.75,A -85,B 0,C 180,E1 -27417.836,E2 -27417.836} C_VEL
LIN {X 0,Y 88.889,Z 336.989,A -85,B 0,C 180,E1 -27424.231,E2 -27424.231} C_VEL
LIN {X 0,Y 86.719,Z 340.933,A -85,B 0,C 180,E1 -27431.091,E2 -27431.091} C_VEL
LIN {X 0,Y 85.954,Z 343.825,A -85,B 0,C 180,E1 -27438.865,E2 -27438.865} C_VEL
LIN {X 0,Y 86.655,Z 345.23,A -85,B 0,C 180,E1 -27445.354,E2 -27445.354} C_VEL
LIN {X 0,Y 87.905,Z 345.701,A -85,B 0,C 180,E1 -27450.006,E2 -27450.006} C_VEL
LIN {X 0,Y 89.664,Z 345.626,A -85,B 0,C 180,E1 -27454.501,E2 -27454.501} C_VEL
LIN {X 0,Y 91.167,Z 344.988,A -85,B 0,C 180,E1 -27458.875,E2 -27458.875} C_VEL
LIN {X 0,Y 92.564,Z 343.917,A -85,B 0,C 180,E1 -27463.032,E2 -27463.032} C_VEL
LIN {X 0,Y 93.521,Z 350.782,A -85,B 0,C 180,E1 -27472.076,E2 -27472.076} C_VEL
LIN {X 0,Y 97.01,Z 356.314,A -85,B 0,C 180,E1 -27480.478,E2 -27480.478} C_VEL
LIN {X 0,Y 102.954,Z 360.974,A -85,B 0,C 180,E1 -27487.912,E2 -27487.912} C_VEL
LIN {X 0,Y 110.688,Z 364.694,A -85,B 0,C 180,E1 -27494.307,E2 -27494.307} C_VEL
LIN {X 0,Y 113.551,Z 365.589,A -85,B 0,C 180,E1 -27497.092,E2 -27497.092} C_VEL
LIN {X 0,Y 103.038,Z 358.514,A -85,B 0,C 180,E1 -27504.566,E2 -27504.566} C_VEL
LIN {X 0,Y 96.138,Z 351.216,A -85,B 0,C 180,E1 -27512.154,E2 -27512.154} C_VEL
LIN {X 0,Y 91.648,Z 342.379,A -85,B 0,C 180,E1 -27520.979,E2 -27520.979} C_VEL
LIN {X 0,Y 89.954,Z 335.09,A -85,B 0,C 180,E1 -27527.593,E2 -27527.593} C_VEL
LIN {X 0,Y 89.066,Z 326.351,A -85,B 0,C 180,E1 -27534.34,E2 -27534.34} C_VEL
LIN {X 0,Y 88.746,Z 316.566,A -85,B 0,C 180,E1 -27540.567,E2 -27540.567} C_VEL
LIN {X 0,Y 88.91,Z 305.677,A -85,B 0,C 180,E1 -27546.24,E2 -27546.24} C_VEL
LIN {X 0,Y 89.572,Z 293.757,A -85,B 0,C 180,E1 -27551.312,E2 -27551.312} C_VEL
LIN {X 0,Y 90.261,Z 284.084,A -85,B 0,C 180,E1 -27554.659,E2 -27554.659} C_VEL
LIN {X 0,Y 89.575,Z 280.208,A -85,B 0,C 180,E1 -27555.647,E2 -27555.647} C_VEL
LIN {X 0,Y 89.583,Z 280.87,A -85,B 0,C 180,E1 -27557.031,E2 -27557.031} C_VEL
LIN {X 0,Y 89.742,Z 281.275,A -85,B 0,C 180,E1 -27558.256,E2 -27558.256} C_VEL
LIN {X 0,Y 92.76,Z 278.984,A -85,B 0,C 180,E1 -27562.261,E2 -27562.261} C_VEL
LIN {X 0,Y 94.307,Z 278.061,A -85,B 0,C 180,E1 -27564.197,E2 -27564.197} C_VEL
LIN {X 0,Y 96.444,Z 276.208,A -85,B 0,C 180,E1 -27565.927,E2 -27565.927} C_VEL
LIN {X 0,Y 99.697,Z 275.007,A -85,B 0,C 180,E1 -27569.568,E2 -27569.568} C_VEL
LIN {X 0,Y 103.758,Z 275.042,A -85,B 0,C 180,E1 -27574.266,E2 -27574.266} C_VEL
LIN {X 0,Y 104.955,Z 275.665,A -85,B 0,C 180,E1 -27575.819,E2 -27575.819} C_VEL
LIN {X 0,Y 105.567,Z 277.69,A -85,B 0,C 180,E1 -27577.596,E2 -27577.596} C_VEL
LIN {X 0,Y 105.52,Z 279.903,A -85,B 0,C 180,E1 -27578.936,E2 -27578.936} C_VEL
LIN {X 0,Y 104.323,Z 287.091,A -85,B 0,C 180,E1 -27582.958,E2 -27582.958} C_VEL
LIN {X 0,Y 104.307,Z 287.925,A -85,B 0,C 180,E1 -27583.614,E2 -27583.614} C_VEL
LIN {X 0,Y 104.045,Z 292.039,A -85,B 0,C 180,E1 -27586.593,E2 -27586.593} C_VEL
LIN {X 0,Y 103.134,Z 296.138,A -85,B 0,C 180,E1 -27589.54,E2 -27589.54} C_VEL
LIN {X 0,Y 99.063,Z 302.268,A -85,B 0,C 180,E1 -27592.907,E2 -27592.907} C_VEL
LIN {X 0,Y 94.177,Z 308.297,A -85,B 0,C 180,E1 -27597.24,E2 -27597.24} C_VEL
LIN {X 0,Y 90.086,Z 312.995,A -85,B 0,C 180,E1 -27602.084,E2 -27602.084} C_VEL
LIN {X 0,Y 86.508,Z 317.122,A -85,B 0,C 180,E1 -27608.55,E2 -27608.55} C_VEL
LIN {X 0,Y 83.374,Z 320.039,A -85,B 0,C 180,E1 -27615.345,E2 -27615.345} C_VEL
LIN {X 0,Y 82.13,Z 321.267,A -85,B 0,C 180,E1 -27620.139,E2 -27620.139} C_VEL
LIN {X 0,Y 81.275,Z 322.015,A -85,B 0,C 180,E1 -27625.033,E2 -27625.033} C_VEL
LIN {X 0,Y 80.972,Z 322.293,A -85,B 0,C 180,E1 -27629.994,E2 -27629.994} C_VEL
LIN {X 0,Y 81.273,Z 322.045,A -85,B 0,C 180,E1 -27634.954,E2 -27634.954} C_VEL
LIN {X 0,Y 82.127,Z 321.335,A -85,B 0,C 180,E1 -27639.848,E2 -27639.848} C_VEL
LIN {X 0,Y 83.369,Z 320.126,A -85,B 0,C 180,E1 -27644.643,E2 -27644.643} C_VEL
LIN {X 0,Y 86.488,Z 317.273,A -85,B 0,C 180,E1 -27651.442,E2 -27651.442} C_VEL
LIN {X 0,Y 90.034,Z 313.193,A -85,B 0,C 180,E1 -27657.921,E2 -27657.921} C_VEL
LIN {X 0,Y 91.817,Z 311.436,A -85,B 0,C 180,E1 -27659.83,E2 -27659.83} C_VEL
LIN {X 0,Y 95.093,Z 307.466,A -85,B 0,C 180,E1 -27663.655,E2 -27663.655} C_VEL
LIN {X 0,Y 100.05,Z 301.159,A -85,B 0,C 180,E1 -27667.919,E2 -27667.919} C_VEL
LIN {X 0,Y 103.216,Z 296.35,A -85,B 0,C 180,E1 -27670.563,E2 -27670.563} C_VEL
LIN {X 0,Y 104.321,Z 291.137,A -85,B 0,C 180,E1 -27674.247,E2 -27674.247} C_VEL
LIN {X 0,Y 104.332,Z 286.568,A -85,B 0,C 180,E1 -27677.807,E2 -27677.807} C_VEL
LIN {X 0,Y 103.438,Z 281.324,A -85,B 0,C 180,E1 -27682.302,E2 -27682.302} C_VEL
LIN {X 0,Y 102.159,Z 277.025,A -85,B 0,C 180,E1 -27686.608,E2 -27686.608} C_VEL
LIN {X 0,Y 100.779,Z 273.397,A -85,B 0,C 180,E1 -27690.78,E2 -27690.78} C_VEL
LIN {X 0,Y 99.427,Z 270.446,A -85,B 0,C 180,E1 -27694.905,E2 -27694.905} C_VEL
LIN {X 0,Y 97.035,Z 266.578,A -85,B 0,C 180,E1 -27703.159,E2 -27703.159} C_VEL
LIN {X 0,Y 95.754,Z 264.692,A -85,B 0,C 180,E1 -27711.559,E2 -27711.559} C_VEL
LIN {X 0,Y 95.724,Z 264.071,A -85,B 0,C 180,E1 -27715.789,E2 -27715.789} C_VEL
LIN {X 0,Y 95.86,Z 264.495,A -85,B 0,C 180,E1 -27720,E2 -27720} C_VEL
LIN {X 0,Y 96.562,Z 268.609,A -85,B 0,C 180,E1 -27728.37,E2 -27728.37} C_VEL
LIN {X 0,Y 97.549,Z 270.828,A -85,B 0,C 180,E1 -27732.482,E2 -27732.482} C_VEL
LIN {X 0,Y 98.098,Z 272.27,A -85,B 0,C 180,E1 -27734.522,E2 -27734.522} C_VEL
LIN {X 0,Y 100.391,Z 278.467,A -85,B 0,C 180,E1 -27741.563,E2 -27741.563} C_VEL
LIN {X 0,Y 102.148,Z 284.221,A -85,B 0,C 180,E1 -27746.577,E2 -27746.577} C_VEL
LIN {X 0,Y 103.388,Z 289.773,A -85,B 0,C 180,E1 -27750.652,E2 -27750.652} C_VEL
LIN {X 0,Y 104.245,Z 295.32,A -85,B 0,C 180,E1 -27754.36,E2 -27754.36} C_VEL
LIN {X 0,Y 104.278,Z 296.713,A -85,B 0,C 180,E1 -27755.206,E2 -27755.206} C_VEL
LIN {X 0,Y 101.213,Z 304.468,A -85,B 0,C 180,E1 -27758.152,E2 -27758.152} C_VEL
LIN {X 0,Y 98.122,Z 311.22,A -85,B 0,C 180,E1 -27761.239,E2 -27761.239} C_VEL
LIN {X 0,Y 94.355,Z 318.022,A -85,B 0,C 180,E1 -27764.968,E2 -27764.968} C_VEL
LIN {X 0,Y 90.289,Z 325.129,A -85,B 0,C 180,E1 -27770.054,E2 -27770.054} C_VEL
LIN {X 0,Y 88.726,Z 327.749,A -85,B 0,C 180,E1 -27772.382,E2 -27772.382} C_VEL
LIN {X 0,Y 84.95,Z 332.659,A -85,B 0,C 180,E1 -27777.477,E2 -27777.477} C_VEL
LIN {X 0,Y 81.446,Z 337.432,A -85,B 0,C 180,E1 -27784.448,E2 -27784.448} C_VEL
LIN {X 0,Y 79.936,Z 339.933,A -85,B 0,C 180,E1 -27789.417,E2 -27789.417} C_VEL
LIN {X 0,Y 78.894,Z 342.993,A -85,B 0,C 180,E1 -27798.492,E2 -27798.492} C_VEL
LIN {X 0,Y 79.476,Z 344.232,A -85,B 0,C 180,E1 -27804.933,E2 -27804.933} C_VEL
LIN {X 0,Y 80.702,Z 344.702,A -85,B 0,C 180,E1 -27810.006,E2 -27810.006} C_VEL
LIN {X 0,Y 82.506,Z 344.63,A -85,B 0,C 180,E1 -27814.893,E2 -27814.893} C_VEL
LIN {X 0,Y 84.202,Z 344.009,A -85,B 0,C 180,E1 -27819.616,E2 -27819.616} C_VEL
LIN {X 0,Y 86.783,Z 342.146,A -85,B 0,C 180,E1 -27826.472,E2 -27826.472} C_VEL
LIN {X 0,Y 88.517,Z 348.83,A -85,B 0,C 180,E1 -27835.899,E2 -27835.899} C_VEL
LIN {X 0,Y 94.499,Z 355.687,A -85,B 0,C 180,E1 -27846.517,E2 -27846.517} C_VEL
LIN {X 0,Y 103.683,Z 361.062,A -85,B 0,C 180,E1 -27855.116,E2 -27855.116} C_VEL
LIN {X 0,Y 104.646,Z 361.492,A -85,B 0,C 180,E1 -27855.823,E2 -27855.823} C_VEL
LIN {X 0,Y 103.985,Z 360.873,A -85,B 0,C 180,E1 -27857.478,E2 -27857.478} C_VEL
LIN {X 0,Y 95.789,Z 354.456,A -85,B 0,C 180,E1 -27864.059,E2 -27864.059} C_VEL
LIN {X 0,Y 88.679,Z 345.809,A -85,B 0,C 180,E1 -27872.89,E2 -27872.89} C_VEL
LIN {X 0,Y 84.901,Z 336.741,A -85,B 0,C 180,E1 -27881.916,E2 -27881.916} C_VEL
LIN {X 0,Y 83.328,Z 328.568,A -85,B 0,C 180,E1 -27889.061,E2 -27889.061} C_VEL
LIN {X 0,Y 82.648,Z 320.462,A -85,B 0,C 180,E1 -27895.122,E2 -27895.122} C_VEL
LIN {X 0,Y 82.323,Z 310.605,A -85,B 0,C 180,E1 -27901.223,E2 -27901.223} C_VEL
LIN {X 0,Y 82.454,Z 301.184,A -85,B 0,C 180,E1 -27906.116,E2 -27906.116} C_VEL
LIN {X 0,Y 83.045,Z 289.081,A -85,B 0,C 180,E1 -27911.441,E2 -27911.441} C_VEL
LIN {X 0,Y 82.804,Z 289.569,A -85,B 0,C 180,E1 -27912.251,E2 -27912.251} C_VEL
LIN {X 0,Y 83.29,Z 289.472,A -85,B 0,C 180,E1 -27914.664,E2 -27914.664} C_VEL
LIN {X 0,Y 84.87,Z 287.986,A -85,B 0,C 180,E1 -27916.848,E2 -27916.848} C_VEL
LIN {X 0,Y 90.848,Z 284.294,A -85,B 0,C 180,E1 -27925.182,E2 -27925.182} C_VEL
LIN {X 0,Y 96.581,Z 281.185,A -85,B 0,C 180,E1 -27930.623,E2 -27930.623} C_VEL
LIN {X 0,Y 103.179,Z 281.233,A -85,B 0,C 180,E1 -27937.81,E2 -27937.81} C_VEL
LIN {X 0,Y 103.863,Z 284.125,A -85,B 0,C 180,E1 -27940.506,E2 -27940.506} C_VEL
LIN {X 0,Y 104.307,Z 287.925,A -85,B 0,C 180,E1 -27943.614,E2 -27943.614} C_VEL
LIN {X 0,Y 103.895,Z 290.047,A -85,B 0,C 180,E1 -27944.941,E2 -27944.941} C_VEL
LIN {X 0,Y 102.09,Z 293.383,A -85,B 0,C 180,E1 -27946.337,E2 -27946.337} C_VEL
LIN {X 0,Y 95.428,Z 301.084,A -85,B 0,C 180,E1 -27949.08,E2 -27949.08} C_VEL
LIN {X 0,Y 93.91,Z 302.845,A -85,B 0,C 180,E1 -27950.036,E2 -27950.036} C_VEL
LIN {X 0,Y 88.349,Z 309.298,A -85,B 0,C 180,E1 -27954.773,E2 -27954.773} C_VEL
LIN {X 0,Y 83.938,Z 313.979,A -85,B 0,C 180,E1 -27959.836,E2 -27959.836} C_VEL
LIN {X 0,Y 80.007,Z 318.102,A -85,B 0,C 180,E1 -27966.709,E2 -27966.709} C_VEL
LIN {X 0,Y 76.595,Z 321.012,A -85,B 0,C 180,E1 -27974.015,E2 -27974.015} C_VEL
LIN {X 0,Y 75.216,Z 322.242,A -85,B 0,C 180,E1 -27979.223,E2 -27979.223} C_VEL
LIN {X 0,Y 74.276,Z 322.989,A -85,B 0,C 180,E1 -27984.564,E2 -27984.564} C_VEL
LIN {X 0,Y 73.944,Z 323.267,A -85,B 0,C 180,E1 -27989.993,E2 -27989.993} C_VEL
LIN {X 0,Y 74.274,Z 323.018,A -85,B 0,C 180,E1 -27995.423,E2 -27995.423} C_VEL
LIN {X 0,Y 75.212,Z 322.309,A -85,B 0,C 180,E1 -28000.764,E2 -28000.764} C_VEL
LIN {X 0,Y 76.59,Z 321.099,A -85,B 0,C 180,E1 -28005.972,E2 -28005.972} C_VEL
LIN {X 0,Y 79.987,Z 318.25,A -85,B 0,C 180,E1 -28013.283,E2 -28013.283} C_VEL
LIN {X 0,Y 83.886,Z 314.173,A -85,B 0,C 180,E1 -28020.17,E2 -28020.17} C_VEL
LIN {X 0,Y 85.791,Z 312.42,A -85,B 0,C 180,E1 -28022.166,E2 -28022.166} C_VEL
LIN {X 0,Y 89.329,Z 308.461,A -85,B 0,C 180,E1 -28026.154,E2 -28026.154} C_VEL
LIN {X 0,Y 94.609,Z 302.176,A -85,B 0,C 180,E1 -28030.533,E2 -28030.533} C_VEL
LIN {X 0,Y 97.58,Z 298.02,A -85,B 0,C 180,E1 -28032.933,E2 -28032.933} C_VEL
LIN {X 0,Y 98.809,Z 293.116,A -85,B 0,C 180,E1 -28036.799,E2 -28036.799} C_VEL
LIN {X 0,Y 98.782,Z 289.323,A -85,B 0,C 180,E1 -28040.184,E2 -28040.184} C_VEL
LIN {X 0,Y 98.422,Z 285.743,A -85,B 0,C 180,E1 -28043.652,E2 -28043.652} C_VEL
LIN {X 0,Y 97.709,Z 282.443,A -85,B 0,C 180,E1 -28047.353,E2 -28047.353} C_VEL
LIN {X 0,Y 96.75,Z 279.115,A -85,B 0,C 180,E1 -28051.588,E2 -28051.588} C_VEL
LIN {X 0,Y 95.655,Z 276.174,A -85,B 0,C 180,E1 -28056.165,E2 -28056.165} C_VEL
LIN {X 0,Y 94.207,Z 273.37,A -85,B 0,C 180,E1 -28062.638,E2 -28062.638} C_VEL
LIN {X 0,Y 93.148,Z 271.355,A -85,B 0,C 180,E1 -28071.321,E2 -28071.321} C_VEL
LIN {X 0,Y 93.225,Z 270.752,A -85,B 0,C 180,E1 -28075.676,E2 -28075.676} C_VEL
LIN {X 0,Y 93.306,Z 271.348,A -85,B 0,C 180,E1 -28080,E2 -28080} C_VEL
LIN {X 0,Y 94.187,Z 276.549,A -85,B 0,C 180,E1 -28090.751,E2 -28090.751} C_VEL
LIN {X 0,Y 94.628,Z 277.856,A -85,B 0,C 180,E1 -28092.874,E2 -28092.874} C_VEL
LIN {X 0,Y 96.327,Z 283.854,A -85,B 0,C 180,E1 -28100.277,E2 -28100.277} C_VEL
LIN {X 0,Y 97.593,Z 289.472,A -85,B 0,C 180,E1 -28105.6,E2 -28105.6} C_VEL
LIN {X 0,Y 98.477,Z 296.43,A -85,B 0,C 180,E1 -28111.096,E2 -28111.096} C_VEL
LIN {X 0,Y 98.526,Z 299.348,A -85,B 0,C 180,E1 -28113.066,E2 -28113.066} C_VEL
LIN {X 0,Y 93.794,Z 309.367,A -85,B 0,C 180,E1 -28117.403,E2 -28117.403} C_VEL
LIN {X 0,Y 89.303,Z 316.954,A -85,B 0,C 180,E1 -28121.624,E2 -28121.624} C_VEL
LIN {X 0,Y 84.788,Z 324.077,A -85,B 0,C 180,E1 -28126.865,E2 -28126.865} C_VEL
LIN {X 0,Y 82.559,Z 327.423,A -85,B 0,C 180,E1 -28130.009,E2 -28130.009} C_VEL
LIN {X 0,Y 77.525,Z 333.394,A -85,B 0,C 180,E1 -28137.057,E2 -28137.057} C_VEL
LIN {X 0,Y 74.052,Z 337.754,A -85,B 0,C 180,E1 -28144.726,E2 -28144.726} C_VEL
LIN {X 0,Y 72.177,Z 340.859,A -85,B 0,C 180,E1 -28153.023,E2 -28153.023} C_VEL
LIN {X 0,Y 71.844,Z 342.312,A -85,B 0,C 180,E1 -28158.725,E2 -28158.725} C_VEL
LIN {X 0,Y 72.297,Z 343.232,A -85,B 0,C 180,E1 -28164.429,E2 -28164.429} C_VEL
LIN {X 0,Y 73.511,Z 343.706,A -85,B 0,C 180,E1 -28170.007,E2 -28170.007} C_VEL
LIN {X 0,Y 75.367,Z 343.637,A -85,B 0,C 180,E1 -28175.358,E2 -28175.358} C_VEL
LIN {X 0,Y 77.242,Z 343.029,A -85,B 0,C 180,E1 -28180.492,E2 -28180.492} C_VEL
LIN {X 0,Y 80.598,Z 340.505,A -85,B 0,C 180,E1 -28189.093,E2 -28189.093} C_VEL
LIN {X 0,Y 81.399,Z 340.121,A -85,B 0,C 180,E1 -28190.21,E2 -28190.21} C_VEL
LIN {X 0,Y 84.029,Z 346.758,A -85,B 0,C 180,E1 -28200.128,E2 -28200.128} C_VEL
LIN {X 0,Y 91.284,Z 353.699,A -85,B 0,C 180,E1 -28210.882,E2 -28210.882} C_VEL
LIN {X 0,Y 95.152,Z 356.085,A -85,B 0,C 180,E1 -28214.569,E2 -28214.569} C_VEL
LIN {X 0,Y 96.819,Z 356.892,A -85,B 0,C 180,E1 -28216.405,E2 -28216.405} C_VEL
LIN {X 0,Y 88.679,Z 349.847,A -85,B 0,C 180,E1 -28223.531,E2 -28223.531} C_VEL
LIN {X 0,Y 82.392,Z 341.527,A -85,B 0,C 180,E1 -28232.021,E2 -28232.021} C_VEL
LIN {X 0,Y 78.616,Z 331.801,A -85,B 0,C 180,E1 -28241.767,E2 -28241.767} C_VEL
LIN {X 0,Y 77.033,Z 322.893,A -85,B 0,C 180,E1 -28249.487,E2 -28249.487} C_VEL
LIN {X 0,Y 76.393,Z 315.792,A -85,B 0,C 180,E1 -28254.722,E2 -28254.722} C_VEL
LIN {X 0,Y 76.053,Z 305.253,A -85,B 0,C 180,E1 -28261.324,E2 -28261.324} C_VEL
LIN {X 0,Y 76.005,Z 297.843,A -85,B 0,C 180,E1 -28265.306,E2 -28265.306} C_VEL
LIN {X 0,Y 76.413,Z 297.417,A -85,B 0,C 180,E1 -28270.6,E2 -28270.6} C_VEL
LIN {X 0,Y 78.143,Z 295.669,A -85,B 0,C 180,E1 -28272.994,E2 -28272.994} C_VEL
LIN {X 0,Y 80.363,Z 294.154,A -85,B 0,C 180,E1 -28277.824,E2 -28277.824} C_VEL
LIN {X 0,Y 82.01,Z 292.984,A -85,B 0,C 180,E1 -28280.047,E2 -28280.047} C_VEL
LIN {X 0,Y 92.99,Z 287.207,A -85,B 0,C 180,E1 -28291.941,E2 -28291.941} C_VEL
LIN {X 0,Y 96.326,Z 287.033,A -85,B 0,C 180,E1 -28295.711,E2 -28295.711} C_VEL
LIN {X 0,Y 98.556,Z 287.464,A -85,B 0,C 180,E1 -28298.326,E2 -28298.326} C_VEL
LIN {X 0,Y 98.716,Z 292.031,A -85,B 0,C 180,E1 -28302.585,E2 -28302.585} C_VEL
LIN {X 0,Y 97.95,Z 296.107,A -85,B 0,C 180,E1 -28305.85,E2 -28305.85} C_VEL
LIN {X 0,Y 97.5,Z 297.797,A -85,B 0,C 180,E1 -28307.164,E2 -28307.164} C_VEL
LIN {X 0,Y 93.91,Z 302.845,A -85,B 0,C 180,E1 -28310.036,E2 -28310.036} C_VEL
LIN {X 0,Y 90.563,Z 306.396,A -85,B 0,C 180,E1 -28312.122,E2 -28312.122} C_VEL
LIN {X 0,Y 83.818,Z 311.708,A -85,B 0,C 180,E1 -28315.373,E2 -28315.373} C_VEL
LIN {X 0,Y 77.27,Z 316.177,A -85,B 0,C 180,E1 -28319.527,E2 -28319.527} C_VEL
LIN {X 0,Y 74.401,Z 318.347,A -85,B 0,C 180,E1 -28323.02,E2 -28323.02} C_VEL
LIN {X 0,Y 72.264,Z 320.175,A -85,B 0,C 180,E1 -28327.099,E2 -28327.099} C_VEL
LIN {X 0,Y 69.866,Z 321.986,A -85,B 0,C 180,E1 -28332.428,E2 -28332.428} C_VEL
LIN {X 0,Y 68.324,Z 323.216,A -85,B 0,C 180,E1 -28338.12,E2 -28338.12} C_VEL
LIN {X 0,Y 67.283,Z 323.963,A -85,B 0,C 180,E1 -28343.997,E2 -28343.997} C_VEL
LIN {X 0,Y 66.916,Z 324.241,A -85,B 0,C 180,E1 -28349.992,E2 -28349.992} C_VEL
LIN {X 0,Y 67.281,Z 323.992,A -85,B 0,C 180,E1 -28355.988,E2 -28355.988} C_VEL
LIN {X 0,Y 68.321,Z 323.283,A -85,B 0,C 180,E1 -28361.865,E2 -28361.865} C_VEL
LIN {X 0,Y 69.86,Z 322.072,A -85,B 0,C 180,E1 -28367.558,E2 -28367.558} C_VEL
LIN {X 0,Y 73.583,Z 319.227,A -85,B 0,C 180,E1 -28375.447,E2 -28375.447} C_VEL
LIN {X 0,Y 77.888,Z 315.155,A -85,B 0,C 180,E1 -28382.77,E2 -28382.77} C_VEL
LIN {X 0,Y 79.915,Z 313.408,A -85,B 0,C 180,E1 -28384.856,E2 -28384.856} C_VEL
LIN {X 0,Y 83.759,Z 309.458,A -85,B 0,C 180,E1 -28388.991,E2 -28388.991} C_VEL
LIN {X 0,Y 89.389,Z 303.194,A -85,B 0,C 180,E1 -28393.459,E2 -28393.459} C_VEL
LIN {X 0,Y 92.084,Z 299.745,A -85,B 0,C 180,E1 -28395.564,E2 -28395.564} C_VEL
